LIN {X 0,Y 488.826,Z 251.849,A -85,B 0,C 180,E1 23621.041,E2 23621.041} C_VEL
LIN {X 0,Y 488.773,Z 251.852,A -85,B 0,C 180,E1 23617.658,E2 23617.658} C_VEL
LIN {X 0,Y 488.76,Z 251.853,A -85,B 0,C 180,E1 23614.093,E2 23614.093} C_VEL
LIN {X 0,Y 488.789,Z 251.852,A -85,B 0,C 180,E1 23610.622,E2 23610.622} C_VEL
LIN {X 0,Y 488.787,Z 251.853,A -85,B 0,C 180,E1 23607.273,E2 23607.273} C_VEL
LIN {X 0,Y 488.779,Z 251.938,A -85,B 0,C 180,E1 23606.334,E2 23606.334} C_VEL
LIN {X 0,Y 489.957,Z 255.178,A -85,B 0,C 180,E1 23606.114,E2 23606.114} C_VEL
LIN {X 0,Y 492.29,Z 257.974,A -85,B 0,C 180,E1 23605.77,E2 23605.77} C_VEL
LIN {X 0,Y 494.97,Z 261.991,A -85,B 0,C 180,E1 23605.374,E2 23605.374} C_VEL
LIN {X 0,Y 505.952,Z 279.714,A -85,B 0,C 180,E1 23603.9,E2 23603.9} C_VEL
LIN {X 0,Y 508.929,Z 284.891,A -85,B 0,C 180,E1 23603.527,E2 23603.527} C_VEL
LIN {X 0,Y 506.243,Z 428.401,A -85,B 0,C 180,E1 23601.176,E2 23601.176} C_VEL
LIN {X 0,Y 504.683,Z 530.578,A -85,B 0,C 180,E1 23599.559,E2 23599.559} C_VEL
LIN {X 0,Y 503.855,Z 552.45,A -85,B 0,C 180,E1 23599.012,E2 23599.012} C_VEL
LIN {X 0,Y 502.715,Z 574.756,A -85,B 0,C 180,E1 23598.227,E2 23598.227} C_VEL
LIN {X 0,Y 501.313,Z 596.319,A -85,B 0,C 180,E1 23597.229,E2 23597.229} C_VEL
LIN {X 0,Y 499.603,Z 617.696,A -85,B 0,C 180,E1 23595.974,E2 23595.974} C_VEL
LIN {X 0,Y 497.826,Z 637.974,A -85,B 0,C 180,E1 23594.516,E2 23594.516} C_VEL
LIN {X 0,Y 496.107,Z 656.509,A -85,B 0,C 180,E1 23592.928,E2 23592.928} C_VEL
LIN {X 0,Y 494.361,Z 674.873,A -85,B 0,C 180,E1 23591.079,E2 23591.079} C_VEL
LIN {X 0,Y 492.804,Z 691.473,A -85,B 0,C 180,E1 23589.107,E2 23589.107} C_VEL
LIN {X 0,Y 491.464,Z 706.623,A -85,B 0,C 180,E1 23587.013,E2 23587.013} C_VEL
LIN {X 0,Y 490.28,Z 720.943,A -85,B 0,C 180,E1 23584.681,E2 23584.681} C_VEL
LIN {X 0,Y 489.411,Z 733.128,A -85,B 0,C 180,E1 23582.343,E2 23582.343} C_VEL
LIN {X 0,Y 488.737,Z 744.343,A -85,B 0,C 180,E1 23579.767,E2 23579.767} C_VEL
LIN {X 0,Y 488.322,Z 753.138,A -85,B 0,C 180,E1 23577.302,E2 23577.302} C_VEL
LIN {X 0,Y 488.079,Z 760.481,A -85,B 0,C 180,E1 23574.712,E2 23574.712} C_VEL
LIN {X 0,Y 487.958,Z 765.848,A -85,B 0,C 180,E1 23572.229,E2 23572.229} C_VEL
LIN {X 0,Y 487.912,Z 769.627,A -85,B 0,C 180,E1 23569.732,E2 23569.732} C_VEL
LIN {X 0,Y 487.912,Z 771.838,A -85,B 0,C 180,E1 23567.215,E2 23567.215} C_VEL
LIN {X 0,Y 487.904,Z 772.465,A -85,B 0,C 180,E1 23564.673,E2 23564.673} C_VEL
LIN {X 0,Y 487.91,Z 771.462,A -85,B 0,C 180,E1 23562.1,E2 23562.1} C_VEL
LIN {X 0,Y 487.918,Z 768.918,A -85,B 0,C 180,E1 23559.615,E2 23559.615} C_VEL
LIN {X 0,Y 487.984,Z 764.727,A -85,B 0,C 180,E1 23557.091,E2 23557.091} C_VEL
LIN {X 0,Y 488.128,Z 758.759,A -85,B 0,C 180,E1 23554.525,E2 23554.525} C_VEL
LIN {X 0,Y 488.397,Z 751.272,A -85,B 0,C 180,E1 23552.045,E2 23552.045} C_VEL
LIN {X 0,Y 488.888,Z 741.478,A -85,B 0,C 180,E1 23549.432,E2 23549.432} C_VEL
LIN {X 0,Y 489.602,Z 730.156,A -85,B 0,C 180,E1 23546.96,E2 23546.96} C_VEL
LIN {X 0,Y 490.56,Z 717.417,A -85,B 0,C 180,E1 23544.616,E2 23544.616} C_VEL
LIN {X 0,Y 491.761,Z 702.995,A -85,B 0,C 180,E1 23542.37,E2 23542.37} C_VEL
LIN {X 0,Y 493.172,Z 687.603,A -85,B 0,C 180,E1 23540.313,E2 23540.313} C_VEL
LIN {X 0,Y 494.808,Z 670.219,A -85,B 0,C 180,E1 23538.336,E2 23538.336} C_VEL
LIN {X 0,Y 496.461,Z 652.681,A -85,B 0,C 180,E1 23536.629,E2 23536.629} C_VEL
LIN {X 0,Y 498.323,Z 632.595,A -85,B 0,C 180,E1 23534.982,E2 23534.982} C_VEL
LIN {X 0,Y 500.016,Z 612.711,A -85,B 0,C 180,E1 23533.621,E2 23533.621} C_VEL
LIN {X 0,Y 501.553,Z 593.125,A -85,B 0,C 180,E1 23532.517,E2 23532.517} C_VEL
LIN {X 0,Y 502.952,Z 571.382,A -85,B 0,C 180,E1 23531.536,E2 23531.536} C_VEL
LIN {X 0,Y 503.202,Z 567.217,A -85,B 0,C 180,E1 23531.379,E2 23531.379} C_VEL
LIN {X 0,Y 502.78,Z 559.985,A -85,B 0,C 180,E1 23531.059,E2 23531.059} C_VEL
LIN {X 0,Y 498.556,Z 542.003,A -85,B 0,C 180,E1 23530.149,E2 23530.149} C_VEL
LIN {X 0,Y 497.979,Z 534.584,A -85,B 0,C 180,E1 23529.907,E2 23529.907} C_VEL
LIN {X 0,Y 498.643,Z 507.178,A -85,B 0,C 180,E1 23529.418,E2 23529.418} C_VEL
LIN {X 0,Y 501.545,Z 350.429,A -85,B 0,C 180,E1 23526.864,E2 23526.864} C_VEL
LIN {X 0,Y 502.677,Z 287.585,A -85,B 0,C 180,E1 23525.824,E2 23525.824} C_VEL
LIN {X 0,Y 489.417,Z 266.799,A -85,B 0,C 180,E1 23524.129,E2 23524.129} C_VEL
LIN {X 0,Y 484.118,Z 258.644,A -85,B 0,C 180,E1 23523.414,E2 23523.414} C_VEL
LIN {X 0,Y 481.453,Z 254.949,A -85,B 0,C 180,E1 23523.053,E2 23523.053} C_VEL
LIN {X 0,Y 480.884,Z 252.838,A -85,B 0,C 180,E1 23522.938,E2 23522.938} C_VEL
LIN {X 0,Y 480.896,Z 252.835,A -85,B 0,C 180,E1 23519.386,E2 23519.386} C_VEL
LIN {X 0,Y 480.859,Z 252.836,A -85,B 0,C 180,E1 23515.892,E2 23515.892} C_VEL
LIN {X 0,Y 480.851,Z 252.838,A -85,B 0,C 180,E1 23512.238,E2 23512.238} C_VEL
LIN {X 0,Y 480.877,Z 252.834,A -85,B 0,C 180,E1 23508.676,E2 23508.676} C_VEL
LIN {X 0,Y 480.896,Z 252.833,A -85,B 0,C 180,E1 23505.065,E2 23505.065} C_VEL
LIN {X 0,Y 480.863,Z 252.833,A -85,B 0,C 180,E1 23501.515,E2 23501.515} C_VEL
LIN {X 0,Y 480.847,Z 252.834,A -85,B 0,C 180,E1 23498.009,E2 23498.009} C_VEL
LIN {X 0,Y 480.877,Z 252.835,A -85,B 0,C 180,E1 23494.533,E2 23494.533} C_VEL
LIN {X 0,Y 480.891,Z 252.83,A -85,B 0,C 180,E1 23490.954,E2 23490.954} C_VEL
LIN {X 0,Y 480.848,Z 252.833,A -85,B 0,C 180,E1 23487.498,E2 23487.498} C_VEL
LIN {X 0,Y 480.844,Z 252.834,A -85,B 0,C 180,E1 23483.914,E2 23483.914} C_VEL
LIN {X 0,Y 480.88,Z 252.836,A -85,B 0,C 180,E1 23480.426,E2 23480.426} C_VEL
LIN {X 0,Y 480.875,Z 252.831,A -85,B 0,C 180,E1 23476.902,E2 23476.902} C_VEL
LIN {X 0,Y 480.838,Z 252.834,A -85,B 0,C 180,E1 23473.447,E2 23473.447} C_VEL
LIN {X 0,Y 480.843,Z 252.835,A -85,B 0,C 180,E1 23469.809,E2 23469.809} C_VEL
LIN {X 0,Y 480.887,Z 252.831,A -85,B 0,C 180,E1 23466.343,E2 23466.343} C_VEL
LIN {X 0,Y 480.864,Z 252.835,A -85,B 0,C 180,E1 23462.779,E2 23462.779} C_VEL
LIN {X 0,Y 480.832,Z 252.838,A -85,B 0,C 180,E1 23459.374,E2 23459.374} C_VEL
LIN {X 0,Y 480.854,Z 252.84,A -85,B 0,C 180,E1 23455.846,E2 23455.846} C_VEL
LIN {X 0,Y 480.888,Z 252.831,A -85,B 0,C 180,E1 23452.32,E2 23452.32} C_VEL
LIN {X 0,Y 480.84,Z 252.835,A -85,B 0,C 180,E1 23448.824,E2 23448.824} C_VEL
LIN {X 0,Y 480.83,Z 252.838,A -85,B 0,C 180,E1 23445.326,E2 23445.326} C_VEL
LIN {X 0,Y 480.868,Z 252.841,A -85,B 0,C 180,E1 23441.867,E2 23441.867} C_VEL
LIN {X 0,Y 480.859,Z 252.833,A -85,B 0,C 180,E1 23438.384,E2 23438.384} C_VEL
LIN {X 0,Y 480.823,Z 252.833,A -85,B 0,C 180,E1 23434.877,E2 23434.877} C_VEL
LIN {X 0,Y 480.828,Z 252.836,A -85,B 0,C 180,E1 23431.282,E2 23431.282} C_VEL
LIN {X 0,Y 480.885,Z 252.838,A -85,B 0,C 180,E1 23427.89,E2 23427.89} C_VEL
LIN {X 0,Y 480.84,Z 252.835,A -85,B 0,C 180,E1 23424.311,E2 23424.311} C_VEL
LIN {X 0,Y 480.817,Z 252.836,A -85,B 0,C 180,E1 23420.828,E2 23420.828} C_VEL
LIN {X 0,Y 480.837,Z 252.838,A -85,B 0,C 180,E1 23417.297,E2 23417.297} C_VEL
LIN {X 0,Y 480.87,Z 252.834,A -85,B 0,C 180,E1 23413.832,E2 23413.832} C_VEL
LIN {X 0,Y 480.82,Z 252.836,A -85,B 0,C 180,E1 23410.3,E2 23410.3} C_VEL
LIN {X 0,Y 480.813,Z 252.838,A -85,B 0,C 180,E1 23406.806,E2 23406.806} C_VEL
LIN {X 0,Y 480.853,Z 252.839,A -85,B 0,C 180,E1 23403.336,E2 23403.336} C_VEL
LIN {X 0,Y 480.839,Z 252.836,A -85,B 0,C 180,E1 23399.879,E2 23399.879} C_VEL
LIN {X 0,Y 480.812,Z 252.839,A -85,B 0,C 180,E1 23396.422,E2 23396.422} C_VEL
LIN {X 0,Y 480.834,Z 252.839,A -85,B 0,C 180,E1 23392.951,E2 23392.951} C_VEL
LIN {X 0,Y 480.87,Z 252.837,A -85,B 0,C 180,E1 23389.456,E2 23389.456} C_VEL
LIN {X 0,Y 480.823,Z 252.837,A -85,B 0,C 180,E1 23386.04,E2 23386.04} C_VEL
LIN {X 0,Y 480.821,Z 252.838,A -85,B 0,C 180,E1 23382.45,E2 23382.45} C_VEL
LIN {X 0,Y 480.866,Z 252.834,A -85,B 0,C 180,E1 23378.998,E2 23378.998} C_VEL
LIN {X 0,Y 480.849,Z 252.837,A -85,B 0,C 180,E1 23375.556,E2 23375.556} C_VEL
LIN {X 0,Y 480.822,Z 252.837,A -85,B 0,C 180,E1 23372.097,E2 23372.097} C_VEL
LIN {X 0,Y 480.853,Z 252.837,A -85,B 0,C 180,E1 23368.678,E2 23368.678} C_VEL
LIN {X 0,Y 480.879,Z 252.835,A -85,B 0,C 180,E1 23365.124,E2 23365.124} C_VEL
LIN {X 0,Y 480.837,Z 252.839,A -85,B 0,C 180,E1 23361.62,E2 23361.62} C_VEL
LIN {X 0,Y 480.833,Z 252.842,A -85,B 0,C 180,E1 23358.108,E2 23358.108} C_VEL
LIN {X 0,Y 480.893,Z 252.932,A -85,B 0,C 180,E1 23356.746,E2 23356.746} C_VEL
LIN {X 0,Y 482.026,Z 256.137,A -85,B 0,C 180,E1 23356.311,E2 23356.311} C_VEL
LIN {X 0,Y 486.724,Z 266.041,A -85,B 0,C 180,E1 23354.868,E2 23354.868} C_VEL
LIN {X 0,Y 494.252,Z 282.954,A -85,B 0,C 180,E1 23352.577,E2 23352.577} C_VEL
LIN {X 0,Y 498.97,Z 294.265,A -85,B 0,C 180,E1 23351.153,E2 23351.153} C_VEL
LIN {X 0,Y 498.76,Z 300.518,A -85,B 0,C 180,E1 23350.689,E2 23350.689} C_VEL
LIN {X 0,Y 503.225,Z 328.094,A -85,B 0,C 180,E1 23349.716,E2 23349.716} C_VEL
LIN {X 0,Y 499.682,Z 515.938,A -85,B 0,C 180,E1 23346.648,E2 23346.648} C_VEL
LIN {X 0,Y 498.054,Z 606.169,A -85,B 0,C 180,E1 23345.186,E2 23345.186} C_VEL
LIN {X 0,Y 497.13,Z 628.175,A -85,B 0,C 180,E1 23344.647,E2 23344.647} C_VEL
LIN {X 0,Y 495.947,Z 649.87,A -85,B 0,C 180,E1 23343.911,E2 23343.911} C_VEL
LIN {X 0,Y 494.532,Z 671.447,A -85,B 0,C 180,E1 23342.958,E2 23342.958} C_VEL
LIN {X 0,Y 492.943,Z 691.876,A -85,B 0,C 180,E1 23341.826,E2 23341.826} C_VEL
LIN {X 0,Y 491.226,Z 712.419,A -85,B 0,C 180,E1 23340.451,E2 23340.451} C_VEL
LIN {X 0,Y 489.577,Z 729.553,A -85,B 0,C 180,E1 23339.061,E2 23339.061} C_VEL
LIN {X 0,Y 487.819,Z 746.483,A -85,B 0,C 180,E1 23337.439,E2 23337.439} C_VEL
LIN {X 0,Y 486.065,Z 763.653,A -85,B 0,C 180,E1 23335.526,E2 23335.526} C_VEL
LIN {X 0,Y 484.507,Z 779.487,A -85,B 0,C 180,E1 23333.469,E2 23333.469} C_VEL
LIN {X 0,Y 483.123,Z 794.1,A -85,B 0,C 180,E1 23331.232,E2 23331.232} C_VEL
LIN {X 0,Y 482.039,Z 806.869,A -85,B 0,C 180,E1 23328.941,E2 23328.941} C_VEL
LIN {X 0,Y 481.203,Z 818.27,A -85,B 0,C 180,E1 23326.537,E2 23326.537} C_VEL
LIN {X 0,Y 480.621,Z 827.976,A -85,B 0,C 180,E1 23324.086,E2 23324.086} C_VEL
LIN {X 0,Y 480.255,Z 835.826,A -85,B 0,C 180,E1 23321.649,E2 23321.649} C_VEL
LIN {X 0,Y 480.045,Z 842.385,A -85,B 0,C 180,E1 23319.107,E2 23319.107} C_VEL
LIN {X 0,Y 479.949,Z 847.021,A -85,B 0,C 180,E1 23316.698,E2 23316.698} C_VEL
LIN {X 0,Y 479.913,Z 850.447,A -85,B 0,C 180,E1 23314.061,E2 23314.061} C_VEL
LIN {X 0,Y 479.898,Z 852.21,A -85,B 0,C 180,E1 23311.551,E2 23311.551} C_VEL
LIN {X 0,Y 479.91,Z 852.326,A -85,B 0,C 180,E1 23309.044,E2 23309.044} C_VEL
LIN {X 0,Y 479.909,Z 850.897,A -85,B 0,C 180,E1 23306.415,E2 23306.415} C_VEL
LIN {X 0,Y 479.935,Z 848.137,A -85,B 0,C 180,E1 23304.02,E2 23304.02} C_VEL
LIN {X 0,Y 480.008,Z 843.65,A -85,B 0,C 180,E1 23301.494,E2 23301.494} C_VEL
LIN {X 0,Y 480.176,Z 837.933,A -85,B 0,C 180,E1 23299.076,E2 23299.076} C_VEL
LIN {X 0,Y 480.484,Z 830.473,A -85,B 0,C 180,E1 23296.644,E2 23296.644} C_VEL
LIN {X 0,Y 481.033,Z 820.833,A -85,B 0,C 180,E1 23294.075,E2 23294.075} C_VEL
LIN {X 0,Y 481.779,Z 810.346,A -85,B 0,C 180,E1 23291.736,E2 23291.736} C_VEL
LIN {X 0,Y 482.795,Z 797.753,A -85,B 0,C 180,E1 23289.385,E2 23289.385} C_VEL
LIN {X 0,Y 484.073,Z 783.703,A -85,B 0,C 180,E1 23287.149,E2 23287.149} C_VEL
LIN {X 0,Y 485.611,Z 768.194,A -85,B 0,C 180,E1 23285.033,E2 23285.033} C_VEL
LIN {X 0,Y 487.338,Z 751.503,A -85,B 0,C 180,E1 23283.081,E2 23283.081} C_VEL
LIN {X 0,Y 489.084,Z 734.081,A -85,B 0,C 180,E1 23281.353,E2 23281.353} C_VEL
LIN {X 0,Y 490.931,Z 715.707,A -85,B 0,C 180,E1 23279.797,E2 23279.797} C_VEL
LIN {X 0,Y 492.168,Z 700.762,A -85,B 0,C 180,E1 23278.749,E2 23278.749} C_VEL
LIN {X 0,Y 493.688,Z 680.03,A -85,B 0,C 180,E1 23277.54,E2 23277.54} C_VEL
LIN {X 0,Y 495.09,Z 659.096,A -85,B 0,C 180,E1 23276.54,E2 23276.54} C_VEL
LIN {X 0,Y 496.257,Z 636.725,A -85,B 0,C 180,E1 23275.709,E2 23275.709} C_VEL
LIN {X 0,Y 497.248,Z 614.263,A -85,B 0,C 180,E1 23275.096,E2 23275.096} C_VEL
LIN {X 0,Y 497.876,Z 589.797,A -85,B 0,C 180,E1 23274.643,E2 23274.643} C_VEL
LIN {X 0,Y 500.406,Z 423.697,A -85,B 0,C 180,E1 23272.015,E2 23272.015} C_VEL
LIN {X 0,Y 502.407,Z 326.034,A -85,B 0,C 180,E1 23270.334,E2 23270.334} C_VEL
LIN {X 0,Y 497.215,Z 292.664,A -85,B 0,C 180,E1 23269.123,E2 23269.123} C_VEL
LIN {X 0,Y 488.051,Z 269.345,A -85,B 0,C 180,E1 23266.234,E2 23266.234} C_VEL
LIN {X 0,Y 483.81,Z 259.793,A -85,B 0,C 180,E1 23264.808,E2 23264.808} C_VEL
LIN {X 0,Y 482.417,Z 256.717,A -85,B 0,C 180,E1 23264.305,E2 23264.305} C_VEL
LIN {X 0,Y 480.922,Z 253.362,A -85,B 0,C 180,E1 23263.732,E2 23263.732} C_VEL
LIN {X 0,Y 480.845,Z 252.841,A -85,B 0,C 180,E1 23263.645,E2 23263.645} C_VEL
LIN {X 0,Y 480.825,Z 252.843,A -85,B 0,C 180,E1 23260.139,E2 23260.139} C_VEL
LIN {X 0,Y 480.863,Z 252.84,A -85,B 0,C 180,E1 23256.788,E2 23256.788} C_VEL
LIN {X 0,Y 480.858,Z 252.839,A -85,B 0,C 180,E1 23253.291,E2 23253.291} C_VEL
LIN {X 0,Y 480.818,Z 252.844,A -85,B 0,C 180,E1 23249.87,E2 23249.87} C_VEL
LIN {X 0,Y 480.877,Z 253.089,A -85,B 0,C 180,E1 23247.326,E2 23247.326} C_VEL
LIN {X 0,Y 482.124,Z 256.249,A -85,B 0,C 180,E1 23247.067,E2 23247.067} C_VEL
LIN {X 0,Y 484.497,Z 259.065,A -85,B 0,C 180,E1 23246.672,E2 23246.672} C_VEL
LIN {X 0,Y 487.154,Z 263.069,A -85,B 0,C 180,E1 23246.243,E2 23246.243} C_VEL
LIN {X 0,Y 493.728,Z 273.293,A -85,B 0,C 180,E1 23245.247,E2 23245.247} C_VEL
LIN {X 0,Y 502.608,Z 287.934,A -85,B 0,C 180,E1 23244.046,E2 23244.046} C_VEL
LIN {X 0,Y 499.77,Z 411.695,A -85,B 0,C 180,E1 23241.94,E2 23241.94} C_VEL
LIN {X 0,Y 497.748,Z 532.141,A -85,B 0,C 180,E1 23239.996,E2 23239.996} C_VEL
LIN {X 0,Y 496.86,Z 554.258,A -85,B 0,C 180,E1 23239.428,E2 23239.428} C_VEL
LIN {X 0,Y 495.706,Z 575.864,A -85,B 0,C 180,E1 23238.651,E2 23238.651} C_VEL
LIN {X 0,Y 494.28,Z 596.991,A -85,B 0,C 180,E1 23237.665,E2 23237.665} C_VEL
LIN {X 0,Y 492.582,Z 617.72,A -85,B 0,C 180,E1 23236.45,E2 23236.45} C_VEL
LIN {X 0,Y 490.853,Z 636.705,A -85,B 0,C 180,E1 23235.086,E2 23235.086} C_VEL
LIN {X 0,Y 488.972,Z 655.448,A -85,B 0,C 180,E1 23233.481,E2 23233.481} C_VEL
LIN {X 0,Y 487.012,Z 674.481,A -85,B 0,C 180,E1 23231.548,E2 23231.548} C_VEL
LIN {X 0,Y 485.37,Z 690.695,A -85,B 0,C 180,E1 23229.607,E2 23229.607} C_VEL
LIN {X 0,Y 483.813,Z 706.737,A -85,B 0,C 180,E1 23227.363,E2 23227.363} C_VEL
LIN {X 0,Y 482.52,Z 721.036,A -85,B 0,C 180,E1 23224.994,E2 23224.994} C_VEL
LIN {X 0,Y 481.565,Z 733.206,A -85,B 0,C 180,E1 23222.62,E2 23222.62} C_VEL
LIN {X 0,Y 480.827,Z 744.4,A -85,B 0,C 180,E1 23220.002,E2 23220.002} C_VEL
LIN {X 0,Y 480.368,Z 753.178,A -85,B 0,C 180,E1 23217.496,E2 23217.496} C_VEL
LIN {X 0,Y 480.094,Z 760.514,A -85,B 0,C 180,E1 23214.864,E2 23214.864} C_VEL
LIN {X 0,Y 479.967,Z 765.868,A -85,B 0,C 180,E1 23212.34,E2 23212.34} C_VEL
LIN {X 0,Y 479.912,Z 769.638,A -85,B 0,C 180,E1 23209.802,E2 23209.802} C_VEL
LIN {X 0,Y 479.912,Z 771.885,A -85,B 0,C 180,E1 23207.174,E2 23207.174} C_VEL
LIN {X 0,Y 479.904,Z 772.464,A -85,B 0,C 180,E1 23204.659,E2 23204.659} C_VEL
LIN {X 0,Y 479.91,Z 771.454,A -85,B 0,C 180,E1 23202.042,E2 23202.042} C_VEL
LIN {X 0,Y 479.922,Z 768.906,A -85,B 0,C 180,E1 23199.514,E2 23199.514} C_VEL
LIN {X 0,Y 479.997,Z 764.701,A -85,B 0,C 180,E1 23196.947,E2 23196.947} C_VEL
LIN {X 0,Y 480.151,Z 758.725,A -85,B 0,C 180,E1 23194.336,E2 23194.336} C_VEL
LIN {X 0,Y 480.455,Z 751.222,A -85,B 0,C 180,E1 23191.812,E2 23191.812} C_VEL
LIN {X 0,Y 481.008,Z 741.388,A -85,B 0,C 180,E1 23189.149,E2 23189.149} C_VEL
LIN {X 0,Y 481.796,Z 730.063,A -85,B 0,C 180,E1 23186.639,E2 23186.639} C_VEL
LIN {X 0,Y 482.837,Z 717.379,A -85,B 0,C 180,E1 23184.268,E2 23184.268} C_VEL
LIN {X 0,Y 484.19,Z 702.534,A -85,B 0,C 180,E1 23181.927,E2 23181.927} C_VEL
LIN {X 0,Y 485.697,Z 687.44,A -85,B 0,C 180,E1 23179.887,E2 23179.887} C_VEL
LIN {X 0,Y 487.48,Z 670.032,A -85,B 0,C 180,E1 23177.882,E2 23177.882} C_VEL
LIN {X 0,Y 489.27,Z 652.463,A -85,B 0,C 180,E1 23176.154,E2 23176.154} C_VEL
LIN {X 0,Y 491.276,Z 632.355,A -85,B 0,C 180,E1 23174.487,E2 23174.487} C_VEL
LIN {X 0,Y 493.103,Z 612.202,A -85,B 0,C 180,E1 23173.105,E2 23173.105} C_VEL
LIN {X 0,Y 494.76,Z 591.707,A -85,B 0,C 180,E1 23171.957,E2 23171.957} C_VEL
LIN {X 0,Y 496.194,Z 570.406,A -85,B 0,C 180,E1 23171.005,E2 23171.005} C_VEL
LIN {X 0,Y 497.395,Z 548.543,A -85,B 0,C 180,E1 23170.264,E2 23170.264} C_VEL
LIN {X 0,Y 497.979,Z 534.584,A -85,B 0,C 180,E1 23169.907,E2 23169.907} C_VEL
LIN {X 0,Y 497.434,Z 527.084,A -85,B 0,C 180,E1 23169.683,E2 23169.683} C_VEL
LIN {X 0,Y 492.603,Z 507.384,A -85,B 0,C 180,E1 23168.951,E2 23168.951} C_VEL
LIN {X 0,Y 492.087,Z 500.873,A -85,B 0,C 180,E1 23168.801,E2 23168.801} C_VEL
LIN {X 0,Y 495.963,Z 317.795,A -85,B 0,C 180,E1 23165.755,E2 23165.755} C_VEL
LIN {X 0,Y 496.395,Z 290.909,A -85,B 0,C 180,E1 23165.299,E2 23165.299} C_VEL
LIN {X 0,Y 484.26,Z 271.876,A -85,B 0,C 180,E1 23163.704,E2 23163.704} C_VEL
LIN {X 0,Y 477.954,Z 262.595,A -85,B 0,C 180,E1 23162.844,E2 23162.844} C_VEL
LIN {X 0,Y 475.512,Z 258.789,A -85,B 0,C 180,E1 23162.497,E2 23162.497} C_VEL
LIN {X 0,Y 473.393,Z 255.718,A -85,B 0,C 180,E1 23162.194,E2 23162.194} C_VEL
LIN {X 0,Y 472.921,Z 253.828,A -85,B 0,C 180,E1 23162.087,E2 23162.087} C_VEL
LIN {X 0,Y 472.92,Z 253.828,A -85,B 0,C 180,E1 23158.406,E2 23158.406} C_VEL
LIN {X 0,Y 472.948,Z 253.822,A -85,B 0,C 180,E1 23154.88,E2 23154.88} C_VEL
LIN {X 0,Y 472.96,Z 253.821,A -85,B 0,C 180,E1 23151.193,E2 23151.193} C_VEL
LIN {X 0,Y 472.93,Z 253.823,A -85,B 0,C 180,E1 23147.552,E2 23147.552} C_VEL
LIN {X 0,Y 472.91,Z 253.82,A -85,B 0,C 180,E1 23143.948,E2 23143.948} C_VEL
LIN {X 0,Y 472.922,Z 253.827,A -85,B 0,C 180,E1 23140.354,E2 23140.354} C_VEL
LIN {X 0,Y 472.958,Z 253.823,A -85,B 0,C 180,E1 23136.8,E2 23136.8} C_VEL
LIN {X 0,Y 472.937,Z 253.821,A -85,B 0,C 180,E1 23133.152,E2 23133.152} C_VEL
LIN {X 0,Y 472.906,Z 253.82,A -85,B 0,C 180,E1 23129.638,E2 23129.638} C_VEL
LIN {X 0,Y 472.907,Z 253.817,A -85,B 0,C 180,E1 23126,E2 23126} C_VEL
LIN {X 0,Y 472.946,Z 253.818,A -85,B 0,C 180,E1 23122.47,E2 23122.47} C_VEL
LIN {X 0,Y 472.938,Z 253.821,A -85,B 0,C 180,E1 23118.909,E2 23118.909} C_VEL
LIN {X 0,Y 472.901,Z 253.823,A -85,B 0,C 180,E1 23115.429,E2 23115.429} C_VEL
LIN {X 0,Y 472.904,Z 253.824,A -85,B 0,C 180,E1 23111.766,E2 23111.766} C_VEL
LIN {X 0,Y 472.946,Z 253.827,A -85,B 0,C 180,E1 23108.288,E2 23108.288} C_VEL
LIN {X 0,Y 472.933,Z 253.821,A -85,B 0,C 180,E1 23104.721,E2 23104.721} C_VEL
LIN {X 0,Y 472.897,Z 253.822,A -85,B 0,C 180,E1 23101.181,E2 23101.181} C_VEL
LIN {X 0,Y 472.896,Z 253.821,A -85,B 0,C 180,E1 23097.519,E2 23097.519} C_VEL
LIN {X 0,Y 472.928,Z 253.823,A -85,B 0,C 180,E1 23094.005,E2 23094.005} C_VEL
LIN {X 0,Y 472.934,Z 253.826,A -85,B 0,C 180,E1 23090.481,E2 23090.481} C_VEL
LIN {X 0,Y 472.891,Z 253.827,A -85,B 0,C 180,E1 23087.014,E2 23087.014} C_VEL
LIN {X 0,Y 472.891,Z 253.826,A -85,B 0,C 180,E1 23083.339,E2 23083.339} C_VEL
LIN {X 0,Y 472.927,Z 253.822,A -85,B 0,C 180,E1 23079.833,E2 23079.833} C_VEL
LIN {X 0,Y 472.924,Z 253.828,A -85,B 0,C 180,E1 23076.294,E2 23076.294} C_VEL
LIN {X 0,Y 472.886,Z 253.828,A -85,B 0,C 180,E1 23072.768,E2 23072.768} C_VEL
LIN {X 0,Y 472.884,Z 253.826,A -85,B 0,C 180,E1 23069.096,E2 23069.096} C_VEL
LIN {X 0,Y 472.926,Z 253.821,A -85,B 0,C 180,E1 23065.682,E2 23065.682} C_VEL
LIN {X 0,Y 472.917,Z 253.826,A -85,B 0,C 180,E1 23062.104,E2 23062.104} C_VEL
LIN {X 0,Y 472.878,Z 253.827,A -85,B 0,C 180,E1 23058.617,E2 23058.617} C_VEL
LIN {X 0,Y 472.878,Z 253.826,A -85,B 0,C 180,E1 23054.928,E2 23054.928} C_VEL
LIN {X 0,Y 472.917,Z 253.825,A -85,B 0,C 180,E1 23051.461,E2 23051.461} C_VEL
LIN {X 0,Y 472.911,Z 253.829,A -85,B 0,C 180,E1 23047.897,E2 23047.897} C_VEL
LIN {X 0,Y 472.871,Z 253.828,A -85,B 0,C 180,E1 23044.485,E2 23044.485} C_VEL
LIN {X 0,Y 472.878,Z 253.825,A -85,B 0,C 180,E1 23040.846,E2 23040.846} C_VEL
LIN {X 0,Y 472.929,Z 253.824,A -85,B 0,C 180,E1 23037.454,E2 23037.454} C_VEL
LIN {X 0,Y 472.892,Z 253.825,A -85,B 0,C 180,E1 23033.93,E2 23033.93} C_VEL
LIN {X 0,Y 472.877,Z 253.828,A -85,B 0,C 180,E1 23030.383,E2 23030.383} C_VEL
LIN {X 0,Y 472.896,Z 253.825,A -85,B 0,C 180,E1 23026.799,E2 23026.799} C_VEL
LIN {X 0,Y 472.931,Z 253.823,A -85,B 0,C 180,E1 23023.415,E2 23023.415} C_VEL
LIN {X 0,Y 472.893,Z 253.827,A -85,B 0,C 180,E1 23019.84,E2 23019.84} C_VEL
LIN {X 0,Y 472.885,Z 253.825,A -85,B 0,C 180,E1 23016.276,E2 23016.276} C_VEL
LIN {X 0,Y 472.922,Z 253.823,A -85,B 0,C 180,E1 23012.826,E2 23012.826} C_VEL
LIN {X 0,Y 472.921,Z 253.828,A -85,B 0,C 180,E1 23009.367,E2 23009.367} C_VEL
LIN {X 0,Y 472.888,Z 253.83,A -85,B 0,C 180,E1 23005.922,E2 23005.922} C_VEL
LIN {X 0,Y 472.896,Z 253.826,A -85,B 0,C 180,E1 23002.254,E2 23002.254} C_VEL
LIN {X 0,Y 472.947,Z 253.826,A -85,B 0,C 180,E1 22998.815,E2 22998.815} C_VEL
LIN {X 0,Y 472.912,Z 253.941,A -85,B 0,C 180,E1 22997.588,E2 22997.588} C_VEL
LIN {X 0,Y 474.308,Z 257.409,A -85,B 0,C 180,E1 22997.085,E2 22997.085} C_VEL
LIN {X 0,Y 482.059,Z 273.946,A -85,B 0,C 180,E1 22994.648,E2 22994.648} C_VEL
LIN {X 0,Y 490.751,Z 294.314,A -85,B 0,C 180,E1 22991.931,E2 22991.931} C_VEL
LIN {X 0,Y 492.197,Z 298.048,A -85,B 0,C 180,E1 22991.469,E2 22991.469} C_VEL
LIN {X 0,Y 492.304,Z 300.443,A -85,B 0,C 180,E1 22991.326,E2 22991.326} C_VEL
LIN {X 0,Y 496.987,Z 329.547,A -85,B 0,C 180,E1 22990.275,E2 22990.275} C_VEL
LIN {X 0,Y 492.643,Z 539.067,A -85,B 0,C 180,E1 22986.799,E2 22986.799} C_VEL
LIN {X 0,Y 491.203,Z 608.625,A -85,B 0,C 180,E1 22985.632,E2 22985.632} C_VEL
LIN {X 0,Y 490.172,Z 630.155,A -85,B 0,C 180,E1 22985.073,E2 22985.073} C_VEL
LIN {X 0,Y 488.787,Z 652.65,A -85,B 0,C 180,E1 22984.267,E2 22984.267} C_VEL
LIN {X 0,Y 487.271,Z 673.754,A -85,B 0,C 180,E1 22983.29,E2 22983.29} C_VEL
LIN {X 0,Y 485.608,Z 693.572,A -85,B 0,C 180,E1 22982.156,E2 22982.156} C_VEL
LIN {X 0,Y 483.783,Z 713.671,A -85,B 0,C 180,E1 22980.763,E2 22980.763} C_VEL
LIN {X 0,Y 481.903,Z 732.987,A -85,B 0,C 180,E1 22979.18,E2 22979.18} C_VEL
LIN {X 0,Y 480.419,Z 747.492,A -85,B 0,C 180,E1 22977.786,E2 22977.786} C_VEL
LIN {X 0,Y 478.521,Z 764.665,A -85,B 0,C 180,E1 22975.825,E2 22975.825} C_VEL
LIN {X 0,Y 476.945,Z 779.488,A -85,B 0,C 180,E1 22973.864,E2 22973.864} C_VEL
LIN {X 0,Y 475.467,Z 793.778,A -85,B 0,C 180,E1 22971.645,E2 22971.645} C_VEL
LIN {X 0,Y 474.28,Z 806.552,A -85,B 0,C 180,E1 22969.327,E2 22969.327} C_VEL
LIN {X 0,Y 473.361,Z 817.974,A -85,B 0,C 180,E1 22966.892,E2 22966.892} C_VEL
LIN {X 0,Y 472.719,Z 827.516,A -85,B 0,C 180,E1 22964.451,E2 22964.451} C_VEL
LIN {X 0,Y 472.306,Z 835.472,A -85,B 0,C 180,E1 22961.972,E2 22961.972} C_VEL
LIN {X 0,Y 472.074,Z 842.131,A -85,B 0,C 180,E1 22959.385,E2 22959.385} C_VEL
LIN {X 0,Y 471.964,Z 846.815,A -85,B 0,C 180,E1 22956.934,E2 22956.934} C_VEL
LIN {X 0,Y 471.917,Z 850.333,A -85,B 0,C 180,E1 22954.251,E2 22954.251} C_VEL
LIN {X 0,Y 471.902,Z 852.085,A -85,B 0,C 180,E1 22951.82,E2 22951.82} C_VEL
LIN {X 0,Y 471.902,Z 852.371,A -85,B 0,C 180,E1 22949.27,E2 22949.27} C_VEL
LIN {X 0,Y 471.915,Z 851.234,A -85,B 0,C 180,E1 22946.719,E2 22946.719} C_VEL
LIN {X 0,Y 471.934,Z 848.456,A -85,B 0,C 180,E1 22944.162,E2 22944.162} C_VEL
LIN {X 0,Y 472.014,Z 843.904,A -85,B 0,C 180,E1 22941.472,E2 22941.472} C_VEL
LIN {X 0,Y 472.193,Z 838.246,A -85,B 0,C 180,E1 22939.013,E2 22939.013} C_VEL
LIN {X 0,Y 472.526,Z 830.877,A -85,B 0,C 180,E1 22936.539,E2 22936.539} C_VEL
LIN {X 0,Y 473.12,Z 821.347,A -85,B 0,C 180,E1 22933.927,E2 22933.927} C_VEL
LIN {X 0,Y 473.975,Z 810.346,A -85,B 0,C 180,E1 22931.425,E2 22931.425} C_VEL
LIN {X 0,Y 475.083,Z 797.751,A -85,B 0,C 180,E1 22929.035,E2 22929.035} C_VEL
LIN {X 0,Y 476.474,Z 783.702,A -85,B 0,C 180,E1 22926.764,E2 22926.764} C_VEL
LIN {X 0,Y 478.089,Z 768.7,A -85,B 0,C 180,E1 22924.678,E2 22924.678} C_VEL
LIN {X 0,Y 479.924,Z 752.231,A -85,B 0,C 180,E1 22922.719,E2 22922.719} C_VEL
LIN {X 0,Y 481.487,Z 737.1,A -85,B 0,C 180,E1 22921.198,E2 22921.198} C_VEL
LIN {X 0,Y 483.228,Z 718.362,A -85,B 0,C 180,E1 22919.636,E2 22919.636} C_VEL
LIN {X 0,Y 484.932,Z 697.908,A -85,B 0,C 180,E1 22918.209,E2 22918.209} C_VEL
LIN {X 0,Y 486.556,Z 677.003,A -85,B 0,C 180,E1 22917.004,E2 22917.004} C_VEL
LIN {X 0,Y 488.014,Z 655.408,A -85,B 0,C 180,E1 22915.99,E2 22915.99} C_VEL
LIN {X 0,Y 489.308,Z 632.893,A -85,B 0,C 180,E1 22915.165,E2 22915.165} C_VEL
LIN {X 0,Y 490.297,Z 611.071,A -85,B 0,C 180,E1 22914.59,E2 22914.59} C_VEL
LIN {X 0,Y 490.974,Z 581.066,A -85,B 0,C 180,E1 22914.058,E2 22914.058} C_VEL
LIN {X 0,Y 493.584,Z 430.546,A -85,B 0,C 180,E1 22911.619,E2 22911.619} C_VEL
LIN {X 0,Y 496.073,Z 327.503,A -85,B 0,C 180,E1 22909.787,E2 22909.787} C_VEL
LIN {X 0,Y 491.254,Z 296.385,A -85,B 0,C 180,E1 22908.614,E2 22908.614} C_VEL
LIN {X 0,Y 487.702,Z 289.972,A -85,B 0,C 180,E1 22908.06,E2 22908.06} C_VEL
LIN {X 0,Y 481.638,Z 273.393,A -85,B 0,C 180,E1 22905.913,E2 22905.913} C_VEL
LIN {X 0,Y 476.907,Z 262.437,A -85,B 0,C 180,E1 22904.19,E2 22904.19} C_VEL
LIN {X 0,Y 474.728,Z 257.967,A -85,B 0,C 180,E1 22903.363,E2 22903.363} C_VEL
LIN {X 0,Y 472.988,Z 254.341,A -85,B 0,C 180,E1 22902.637,E2 22902.637} C_VEL
LIN {X 0,Y 472.899,Z 253.831,A -85,B 0,C 180,E1 22902.488,E2 22902.488} C_VEL
LIN {X 0,Y 472.954,Z 253.824,A -85,B 0,C 180,E1 22899.051,E2 22899.051} C_VEL
LIN {X 0,Y 472.912,Z 253.83,A -85,B 0,C 180,E1 22895.403,E2 22895.403} C_VEL
LIN {X 0,Y 472.882,Z 253.833,A -85,B 0,C 180,E1 22891.912,E2 22891.912} C_VEL
LIN {X 0,Y 472.924,Z 254.011,A -85,B 0,C 180,E1 22888.469,E2 22888.469} C_VEL
LIN {X 0,Y 474.124,Z 257.22,A -85,B 0,C 180,E1 22888.175,E2 22888.175} C_VEL
LIN {X 0,Y 476.876,Z 260.202,A -85,B 0,C 180,E1 22887.675,E2 22887.675} C_VEL
LIN {X 0,Y 479.489,Z 264.156,A -85,B 0,C 180,E1 22887.193,E2 22887.193} C_VEL
LIN {X 0,Y 486.263,Z 274.296,A -85,B 0,C 180,E1 22886.063,E2 22886.063} C_VEL
LIN {X 0,Y 495.94,Z 290.404,A -85,B 0,C 180,E1 22884.639,E2 22884.639} C_VEL
LIN {X 0,Y 496.338,Z 291.663,A -85,B 0,C 180,E1 22884.571,E2 22884.571} C_VEL
LIN {X 0,Y 493.016,Z 417.507,A -85,B 0,C 180,E1 22882.36,E2 22882.36} C_VEL
LIN {X 0,Y 490.832,Z 533.669,A -85,B 0,C 180,E1 22880.443,E2 22880.443} C_VEL
LIN {X 0,Y 489.924,Z 555.274,A -85,B 0,C 180,E1 22879.878,E2 22879.878} C_VEL
LIN {X 0,Y 488.754,Z 576.5,A -85,B 0,C 180,E1 22879.107,E2 22879.107} C_VEL
LIN {X 0,Y 487.369,Z 596.593,A -85,B 0,C 180,E1 22878.171,E2 22878.171} C_VEL
LIN {X 0,Y 485.657,Z 616.694,A -85,B 0,C 180,E1 22877,E2 22877} C_VEL
LIN {X 0,Y 483.89,Z 635.556,A -85,B 0,C 180,E1 22875.656,E2 22875.656} C_VEL
LIN {X 0,Y 481.897,Z 654.413,A -85,B 0,C 180,E1 22874.051,E2 22874.051} C_VEL
LIN {X 0,Y 479.893,Z 672.455,A -85,B 0,C 180,E1 22872.21,E2 22872.21} C_VEL
LIN {X 0,Y 478.068,Z 689.015,A -85,B 0,C 180,E1 22870.242,E2 22870.242} C_VEL
LIN {X 0,Y 476.331,Z 705.253,A -85,B 0,C 180,E1 22867.965,E2 22867.965} C_VEL
LIN {X 0,Y 474.96,Z 719.136,A -85,B 0,C 180,E1 22865.68,E2 22865.68} C_VEL
LIN {X 0,Y 473.822,Z 732.167,A -85,B 0,C 180,E1 22863.147,E2 22863.147} C_VEL
LIN {X 0,Y 473.013,Z 743.045,A -85,B 0,C 180,E1 22860.607,E2 22860.607} C_VEL
LIN {X 0,Y 472.462,Z 752.474,A -85,B 0,C 180,E1 22857.94,E2 22857.94} C_VEL
LIN {X 0,Y 472.139,Z 759.944,A -85,B 0,C 180,E1 22855.264,E2 22855.264} C_VEL
LIN {X 0,Y 471.986,Z 765.472,A -85,B 0,C 180,E1 22852.7,E2 22852.7} C_VEL
LIN {X 0,Y 471.917,Z 769.363,A -85,B 0,C 180,E1 22850.12,E2 22850.12} C_VEL
LIN {X 0,Y 471.907,Z 771.786,A -85,B 0,C 180,E1 22847.397,E2 22847.397} C_VEL
LIN {X 0,Y 471.908,Z 772.479,A -85,B 0,C 180,E1 22844.77,E2 22844.77} C_VEL
LIN {X 0,Y 471.909,Z 771.529,A -85,B 0,C 180,E1 22842.11,E2 22842.11} C_VEL
LIN {X 0,Y 471.925,Z 768.967,A -85,B 0,C 180,E1 22839.466,E2 22839.466} C_VEL
LIN {X 0,Y 472.003,Z 764.676,A -85,B 0,C 180,E1 22836.798,E2 22836.798} C_VEL
LIN {X 0,Y 472.177,Z 758.69,A -85,B 0,C 180,E1 22834.14,E2 22834.14} C_VEL
LIN {X 0,Y 472.521,Z 751.17,A -85,B 0,C 180,E1 22831.571,E2 22831.571} C_VEL
LIN {X 0,Y 473.137,Z 741.301,A -85,B 0,C 180,E1 22828.857,E2 22828.857} C_VEL
LIN {X 0,Y 474.001,Z 729.968,A -85,B 0,C 180,E1 22826.308,E2 22826.308} C_VEL
LIN {X 0,Y 475.14,Z 717.295,A -85,B 0,C 180,E1 22823.902,E2 22823.902} C_VEL
LIN {X 0,Y 476.555,Z 703.022,A -85,B 0,C 180,E1 22821.611,E2 22821.611} C_VEL
LIN {X 0,Y 478.252,Z 687.277,A -85,B 0,C 180,E1 22819.447,E2 22819.447} C_VEL
LIN {X 0,Y 480.263,Z 669.109,A -85,B 0,C 180,E1 22817.335,E2 22817.335} C_VEL
LIN {X 0,Y 482.215,Z 651.469,A -85,B 0,C 180,E1 22815.593,E2 22815.593} C_VEL
LIN {X 0,Y 484.257,Z 632.041,A -85,B 0,C 180,E1 22813.977,E2 22813.977} C_VEL
LIN {X 0,Y 486.217,Z 611.639,A -85,B 0,C 180,E1 22812.576,E2 22812.576} C_VEL
LIN {X 0,Y 487.963,Z 590.996,A -85,B 0,C 180,E1 22811.418,E2 22811.418} C_VEL
LIN {X 0,Y 489.513,Z 569.127,A -85,B 0,C 180,E1 22810.448,E2 22810.448} C_VEL
LIN {X 0,Y 490.718,Z 547.668,A -85,B 0,C 180,E1 22809.727,E2 22809.727} C_VEL
LIN {X 0,Y 491.607,Z 524.81,A -85,B 0,C 180,E1 22809.194,E2 22809.194} C_VEL
LIN {X 0,Y 492.087,Z 500.873,A -85,B 0,C 180,E1 22808.801,E2 22808.801} C_VEL
LIN {X 0,Y 491.409,Z 493.306,A -85,B 0,C 180,E1 22808.614,E2 22808.614} C_VEL
LIN {X 0,Y 486.679,Z 473.598,A -85,B 0,C 180,E1 22807.865,E2 22807.865} C_VEL
LIN {X 0,Y 486.203,Z 467.096,A -85,B 0,C 180,E1 22807.705,E2 22807.705} C_VEL
LIN {X 0,Y 490.178,Z 294.151,A -85,B 0,C 180,E1 22804.76,E2 22804.76} C_VEL
LIN {X 0,Y 476.956,Z 273.625,A -85,B 0,C 180,E1 22802.975,E2 22802.975} C_VEL
LIN {X 0,Y 470.422,Z 264.08,A -85,B 0,C 180,E1 22802.045,E2 22802.045} C_VEL
LIN {X 0,Y 467.619,Z 259.796,A -85,B 0,C 180,E1 22801.628,E2 22801.628} C_VEL
LIN {X 0,Y 465.527,Z 256.792,A -85,B 0,C 180,E1 22801.318,E2 22801.318} C_VEL
LIN {X 0,Y 465.019,Z 254.814,A -85,B 0,C 180,E1 22801.212,E2 22801.212} C_VEL
LIN {X 0,Y 465.007,Z 254.813,A -85,B 0,C 180,E1 22797.536,E2 22797.536} C_VEL
LIN {X 0,Y 464.979,Z 254.815,A -85,B 0,C 180,E1 22793.959,E2 22793.959} C_VEL
LIN {X 0,Y 464.977,Z 254.816,A -85,B 0,C 180,E1 22790.256,E2 22790.256} C_VEL
LIN {X 0,Y 464.997,Z 254.811,A -85,B 0,C 180,E1 22786.619,E2 22786.619} C_VEL
LIN {X 0,Y 465.017,Z 254.808,A -85,B 0,C 180,E1 22783.049,E2 22783.049} C_VEL
LIN {X 0,Y 464.99,Z 254.812,A -85,B 0,C 180,E1 22779.407,E2 22779.407} C_VEL
LIN {X 0,Y 464.969,Z 254.809,A -85,B 0,C 180,E1 22775.802,E2 22775.802} C_VEL
LIN {X 0,Y 464.972,Z 254.81,A -85,B 0,C 180,E1 22772.096,E2 22772.096} C_VEL
LIN {X 0,Y 465.003,Z 254.807,A -85,B 0,C 180,E1 22768.523,E2 22768.523} C_VEL
LIN {X 0,Y 465.011,Z 254.803,A -85,B 0,C 180,E1 22764.82,E2 22764.82} C_VEL
LIN {X 0,Y 464.971,Z 254.807,A -85,B 0,C 180,E1 22761.344,E2 22761.344} C_VEL
LIN {X 0,Y 464.963,Z 254.811,A -85,B 0,C 180,E1 22757.71,E2 22757.71} C_VEL
LIN {X 0,Y 464.985,Z 254.81,A -85,B 0,C 180,E1 22754.153,E2 22754.153} C_VEL
LIN {X 0,Y 465.012,Z 254.807,A -85,B 0,C 180,E1 22750.534,E2 22750.534} C_VEL
LIN {X 0,Y 464.977,Z 254.812,A -85,B 0,C 180,E1 22746.962,E2 22746.962} C_VEL
LIN {X 0,Y 464.958,Z 254.815,A -85,B 0,C 180,E1 22743.432,E2 22743.432} C_VEL
LIN {X 0,Y 464.97,Z 254.817,A -85,B 0,C 180,E1 22739.814,E2 22739.814} C_VEL
LIN {X 0,Y 465.005,Z 254.81,A -85,B 0,C 180,E1 22736.308,E2 22736.308} C_VEL
LIN {X 0,Y 464.978,Z 254.809,A -85,B 0,C 180,E1 22732.673,E2 22732.673} C_VEL
LIN {X 0,Y 464.951,Z 254.814,A -85,B 0,C 180,E1 22729.178,E2 22729.178} C_VEL
LIN {X 0,Y 464.962,Z 254.817,A -85,B 0,C 180,E1 22725.552,E2 22725.552} C_VEL
LIN {X 0,Y 464.997,Z 254.819,A -85,B 0,C 180,E1 22721.931,E2 22721.931} C_VEL
LIN {X 0,Y 464.989,Z 254.81,A -85,B 0,C 180,E1 22718.296,E2 22718.296} C_VEL
LIN {X 0,Y 464.95,Z 254.81,A -85,B 0,C 180,E1 22714.738,E2 22714.738} C_VEL
LIN {X 0,Y 464.945,Z 254.813,A -85,B 0,C 180,E1 22711.069,E2 22711.069} C_VEL
LIN {X 0,Y 464.98,Z 254.816,A -85,B 0,C 180,E1 22707.638,E2 22707.638} C_VEL
LIN {X 0,Y 464.994,Z 254.813,A -85,B 0,C 180,E1 22703.96,E2 22703.96} C_VEL
LIN {X 0,Y 464.946,Z 254.814,A -85,B 0,C 180,E1 22700.517,E2 22700.517} C_VEL
LIN {X 0,Y 464.939,Z 254.816,A -85,B 0,C 180,E1 22696.874,E2 22696.874} C_VEL
LIN {X 0,Y 464.974,Z 254.817,A -85,B 0,C 180,E1 22693.427,E2 22693.427} C_VEL
LIN {X 0,Y 464.985,Z 254.813,A -85,B 0,C 180,E1 22689.779,E2 22689.779} C_VEL
LIN {X 0,Y 464.938,Z 254.816,A -85,B 0,C 180,E1 22686.295,E2 22686.295} C_VEL
LIN {X 0,Y 464.934,Z 254.818,A -85,B 0,C 180,E1 22682.71,E2 22682.71} C_VEL
LIN {X 0,Y 464.967,Z 254.818,A -85,B 0,C 180,E1 22679.17,E2 22679.17} C_VEL
LIN {X 0,Y 464.987,Z 254.818,A -85,B 0,C 180,E1 22675.559,E2 22675.559} C_VEL
LIN {X 0,Y 464.944,Z 254.817,A -85,B 0,C 180,E1 22672.088,E2 22672.088} C_VEL
LIN {X 0,Y 464.939,Z 254.815,A -85,B 0,C 180,E1 22668.462,E2 22668.462} C_VEL
LIN {X 0,Y 464.968,Z 254.816,A -85,B 0,C 180,E1 22664.903,E2 22664.903} C_VEL
LIN {X 0,Y 464.995,Z 254.811,A -85,B 0,C 180,E1 22661.312,E2 22661.312} C_VEL
LIN {X 0,Y 464.956,Z 254.815,A -85,B 0,C 180,E1 22657.759,E2 22657.759} C_VEL
LIN {X 0,Y 464.945,Z 254.814,A -85,B 0,C 180,E1 22654.252,E2 22654.252} C_VEL
LIN {X 0,Y 464.983,Z 254.812,A -85,B 0,C 180,E1 22650.782,E2 22650.782} C_VEL
LIN {X 0,Y 464.996,Z 254.814,A -85,B 0,C 180,E1 22647.188,E2 22647.188} C_VEL
LIN {X 0,Y 464.954,Z 254.818,A -85,B 0,C 180,E1 22643.744,E2 22643.744} C_VEL
LIN {X 0,Y 464.955,Z 254.819,A -85,B 0,C 180,E1 22640.145,E2 22640.145} C_VEL
LIN {X 0,Y 464.994,Z 254.97,A -85,B 0,C 180,E1 22638.457,E2 22638.457} C_VEL
LIN {X 0,Y 466.162,Z 258.156,A -85,B 0,C 180,E1 22637.994,E2 22637.994} C_VEL
LIN {X 0,Y 467.316,Z 260.443,A -85,B 0,C 180,E1 22637.625,E2 22637.625} C_VEL
LIN {X 0,Y 474.444,Z 275.483,A -85,B 0,C 180,E1 22635.345,E2 22635.345} C_VEL
LIN {X 0,Y 482.307,Z 293.577,A -85,B 0,C 180,E1 22632.839,E2 22632.839} C_VEL
LIN {X 0,Y 484.77,Z 299.43,A -85,B 0,C 180,E1 22632.119,E2 22632.119} C_VEL
LIN {X 0,Y 486.277,Z 302.467,A -85,B 0,C 180,E1 22631.898,E2 22631.898} C_VEL
LIN {X 0,Y 490.792,Z 331.229,A -85,B 0,C 180,E1 22630.843,E2 22630.843} C_VEL
LIN {X 0,Y 486.095,Z 536.473,A -85,B 0,C 180,E1 22627.374,E2 22627.374} C_VEL
LIN {X 0,Y 484.467,Z 608.157,A -85,B 0,C 180,E1 22626.15,E2 22626.15} C_VEL
LIN {X 0,Y 483.359,Z 629.788,A -85,B 0,C 180,E1 22625.581,E2 22625.581} C_VEL
LIN {X 0,Y 481.918,Z 651.707,A -85,B 0,C 180,E1 22624.787,E2 22624.787} C_VEL
LIN {X 0,Y 480.235,Z 673.414,A -85,B 0,C 180,E1 22623.771,E2 22623.771} C_VEL
LIN {X 0,Y 478.477,Z 693.18,A -85,B 0,C 180,E1 22622.623,E2 22622.623} C_VEL
LIN {X 0,Y 476.515,Z 713.228,A -85,B 0,C 180,E1 22621.215,E2 22621.215} C_VEL
LIN {X 0,Y 474.443,Z 733.201,A -85,B 0,C 180,E1 22619.545,E2 22619.545} C_VEL
LIN {X 0,Y 472.595,Z 750.744,A -85,B 0,C 180,E1 22617.827,E2 22617.827} C_VEL
LIN {X 0,Y 470.743,Z 767.645,A -85,B 0,C 180,E1 22615.878,E2 22615.878} C_VEL
LIN {X 0,Y 469,Z 782.872,A -85,B 0,C 180,E1 22613.76,E2 22613.76} C_VEL
LIN {X 0,Y 467.505,Z 796.738,A -85,B 0,C 180,E1 22611.511,E2 22611.511} C_VEL
LIN {X 0,Y 466.286,Z 809.09,A -85,B 0,C 180,E1 22609.151,E2 22609.151} C_VEL
LIN {X 0,Y 465.357,Z 819.813,A -85,B 0,C 180,E1 22606.731,E2 22606.731} C_VEL
LIN {X 0,Y 464.7,Z 829.266,A -85,B 0,C 180,E1 22604.197,E2 22604.197} C_VEL
LIN {X 0,Y 464.287,Z 836.884,A -85,B 0,C 180,E1 22601.678,E2 22601.678} C_VEL
LIN {X 0,Y 464.046,Z 843.148,A -85,B 0,C 180,E1 22599.048,E2 22599.048} C_VEL
LIN {X 0,Y 463.946,Z 847.685,A -85,B 0,C 180,E1 22596.529,E2 22596.529} C_VEL
LIN {X 0,Y 463.91,Z 850.674,A -85,B 0,C 180,E1 22593.954,E2 22593.954} C_VEL
LIN {X 0,Y 463.903,Z 852.258,A -85,B 0,C 180,E1 22591.357,E2 22591.357} C_VEL
LIN {X 0,Y 463.911,Z 852.303,A -85,B 0,C 180,E1 22588.887,E2 22588.887} C_VEL
LIN {X 0,Y 463.91,Z 850.782,A -85,B 0,C 180,E1 22586.168,E2 22586.168} C_VEL
LIN {X 0,Y 463.942,Z 847.816,A -85,B 0,C 180,E1 22583.564,E2 22583.564} C_VEL
LIN {X 0,Y 464.034,Z 843.396,A -85,B 0,C 180,E1 22581.074,E2 22581.074} C_VEL
LIN {X 0,Y 464.272,Z 837.23,A -85,B 0,C 180,E1 22578.445,E2 22578.445} C_VEL
LIN {X 0,Y 464.673,Z 829.661,A -85,B 0,C 180,E1 22575.927,E2 22575.927} C_VEL
LIN {X 0,Y 465.32,Z 820.316,A -85,B 0,C 180,E1 22573.393,E2 22573.393} C_VEL
LIN {X 0,Y 466.233,Z 809.713,A -85,B 0,C 180,E1 22570.975,E2 22570.975} C_VEL
LIN {X 0,Y 467.389,Z 797.75,A -85,B 0,C 180,E1 22568.673,E2 22568.673} C_VEL
LIN {X 0,Y 468.903,Z 783.7,A -85,B 0,C 180,E1 22566.366,E2 22566.366} C_VEL
LIN {X 0,Y 470.623,Z 768.797,A -85,B 0,C 180,E1 22564.265,E2 22564.265} C_VEL
LIN {X 0,Y 472.047,Z 755.012,A -85,B 0,C 180,E1 22562.67,E2 22562.67} C_VEL
LIN {X 0,Y 473.903,Z 736.46,A -85,B 0,C 180,E1 22560.831,E2 22560.831} C_VEL
LIN {X 0,Y 475.771,Z 717.44,A -85,B 0,C 180,E1 22559.227,E2 22559.227} C_VEL
LIN {X 0,Y 477.542,Z 697.223,A -85,B 0,C 180,E1 22557.8,E2 22557.8} C_VEL
LIN {X 0,Y 479.308,Z 675.917,A -85,B 0,C 180,E1 22556.556,E2 22556.556} C_VEL
LIN {X 0,Y 480.857,Z 654.087,A -85,B 0,C 180,E1 22555.521,E2 22555.521} C_VEL
LIN {X 0,Y 482.265,Z 631.406,A -85,B 0,C 180,E1 22554.686,E2 22554.686} C_VEL
LIN {X 0,Y 483.322,Z 609.08,A -85,B 0,C 180,E1 22554.096,E2 22554.096} C_VEL
LIN {X 0,Y 484.063,Z 577.376,A -85,B 0,C 180,E1 22553.534,E2 22553.534} C_VEL
LIN {X 0,Y 486.705,Z 441.558,A -85,B 0,C 180,E1 22551.281,E2 22551.281} C_VEL
LIN {X 0,Y 489.956,Z 329.692,A -85,B 0,C 180,E1 22549.244,E2 22549.244} C_VEL
LIN {X 0,Y 485.704,Z 300.608,A -85,B 0,C 180,E1 22548.111,E2 22548.111} C_VEL
LIN {X 0,Y 478.696,Z 286.934,A -85,B 0,C 180,E1 22546.888,E2 22546.888} C_VEL
LIN {X 0,Y 474.067,Z 274.58,A -85,B 0,C 180,E1 22545.127,E2 22545.127} C_VEL
LIN {X 0,Y 470.326,Z 266.386,A -85,B 0,C 180,E1 22543.703,E2 22543.703} C_VEL
LIN {X 0,Y 468.766,Z 262.968,A -85,B 0,C 180,E1 22543.044,E2 22543.044} C_VEL
LIN {X 0,Y 466.983,Z 259.226,A -85,B 0,C 180,E1 22542.246,E2 22542.246} C_VEL
LIN {X 0,Y 465.173,Z 255.811,A -85,B 0,C 180,E1 22541.396,E2 22541.396} C_VEL
LIN {X 0,Y 465.009,Z 254.815,A -85,B 0,C 180,E1 22541.145,E2 22541.145} C_VEL
LIN {X 0,Y 464.958,Z 254.819,A -85,B 0,C 180,E1 22537.643,E2 22537.643} C_VEL
LIN {X 0,Y 464.945,Z 254.821,A -85,B 0,C 180,E1 22533.996,E2 22533.996} C_VEL
LIN {X 0,Y 464.951,Z 254.821,A -85,B 0,C 180,E1 22530.356,E2 22530.356} C_VEL
LIN {X 0,Y 464.973,Z 255.044,A -85,B 0,C 180,E1 22529.836,E2 22529.836} C_VEL
LIN {X 0,Y 466.177,Z 258.172,A -85,B 0,C 180,E1 22529.483,E2 22529.483} C_VEL
LIN {X 0,Y 469.218,Z 261.312,A -85,B 0,C 180,E1 22528.824,E2 22528.824} C_VEL
LIN {X 0,Y 471.58,Z 265.15,A -85,B 0,C 180,E1 22528.305,E2 22528.305} C_VEL
LIN {X 0,Y 473.202,Z 267.088,A -85,B 0,C 180,E1 22527.998,E2 22527.998} C_VEL
LIN {X 0,Y 477.225,Z 273.203,A -85,B 0,C 180,E1 22527.235,E2 22527.235} C_VEL
LIN {X 0,Y 482.346,Z 281.082,A -85,B 0,C 180,E1 22526.355,E2 22526.355} C_VEL
LIN {X 0,Y 490.216,Z 294.402,A -85,B 0,C 180,E1 22525.136,E2 22525.136} C_VEL
LIN {X 0,Y 486.691,Z 407.298,A -85,B 0,C 180,E1 22523.078,E2 22523.078} C_VEL
LIN {X 0,Y 483.923,Z 535.316,A -85,B 0,C 180,E1 22520.897,E2 22520.897} C_VEL
LIN {X 0,Y 482.981,Z 556.961,A -85,B 0,C 180,E1 22520.318,E2 22520.318} C_VEL
LIN {X 0,Y 481.807,Z 577.431,A -85,B 0,C 180,E1 22519.563,E2 22519.563} C_VEL
LIN {X 0,Y 480.398,Z 597.25,A -85,B 0,C 180,E1 22518.633,E2 22518.633} C_VEL
LIN {X 0,Y 478.694,Z 616.497,A -85,B 0,C 180,E1 22517.505,E2 22517.505} C_VEL
LIN {X 0,Y 476.815,Z 635.731,A -85,B 0,C 180,E1 22516.133,E2 22516.133} C_VEL
LIN {X 0,Y 474.74,Z 654.646,A -85,B 0,C 180,E1 22514.516,E2 22514.516} C_VEL
LIN {X 0,Y 472.739,Z 671.747,A -85,B 0,C 180,E1 22512.77,E2 22512.77} C_VEL
LIN {X 0,Y 470.721,Z 688.282,A -85,B 0,C 180,E1 22510.775,E2 22510.775} C_VEL
LIN {X 0,Y 468.729,Z 705.369,A -85,B 0,C 180,E1 22508.342,E2 22508.342} C_VEL
LIN {X 0,Y 467.245,Z 719.229,A -85,B 0,C 180,E1 22506.02,E2 22506.02} C_VEL
LIN {X 0,Y 466.006,Z 732.245,A -85,B 0,C 180,E1 22503.446,E2 22503.446} C_VEL
LIN {X 0,Y 465.121,Z 743.103,A -85,B 0,C 180,E1 22500.864,E2 22500.864} C_VEL
LIN {X 0,Y 464.519,Z 752.522,A -85,B 0,C 180,E1 22498.151,E2 22498.151} C_VEL
LIN {X 0,Y 464.165,Z 759.977,A -85,B 0,C 180,E1 22495.43,E2 22495.43} C_VEL
LIN {X 0,Y 463.995,Z 765.493,A -85,B 0,C 180,E1 22492.822,E2 22492.822} C_VEL
LIN {X 0,Y 463.921,Z 769.374,A -85,B 0,C 180,E1 22490.199,E2 22490.199} C_VEL
LIN {X 0,Y 463.906,Z 771.792,A -85,B 0,C 180,E1 22487.429,E2 22487.429} C_VEL
LIN {X 0,Y 463.911,Z 772.494,A -85,B 0,C 180,E1 22484.885,E2 22484.885} C_VEL
LIN {X 0,Y 463.909,Z 771.604,A -85,B 0,C 180,E1 22482.181,E2 22482.181} C_VEL
LIN {X 0,Y 463.928,Z 769.052,A -85,B 0,C 180,E1 22479.436,E2 22479.436} C_VEL
LIN {X 0,Y 464.008,Z 764.907,A -85,B 0,C 180,E1 22476.778,E2 22476.778} C_VEL
LIN {X 0,Y 464.194,Z 758.989,A -85,B 0,C 180,E1 22474.074,E2 22474.074} C_VEL
LIN {X 0,Y 464.574,Z 751.42,A -85,B 0,C 180,E1 22471.415,E2 22471.415} C_VEL
LIN {X 0,Y 465.234,Z 741.638,A -85,B 0,C 180,E1 22468.664,E2 22468.664} C_VEL
LIN {X 0,Y 466.154,Z 730.555,A -85,B 0,C 180,E1 22466.108,E2 22466.108} C_VEL
LIN {X 0,Y 467.456,Z 717.294,A -85,B 0,C 180,E1 22463.538,E2 22463.538} C_VEL
LIN {X 0,Y 469.009,Z 702.888,A -85,B 0,C 180,E1 22461.191,E2 22461.191} C_VEL
LIN {X 0,Y 470.848,Z 687.164,A -85,B 0,C 180,E1 22458.995,E2 22458.995} C_VEL
LIN {X 0,Y 472.939,Z 669.822,A -85,B 0,C 180,E1 22456.935,E2 22456.935} C_VEL
LIN {X 0,Y 475.026,Z 652.126,A -85,B 0,C 180,E1 22455.164,E2 22455.164} C_VEL
LIN {X 0,Y 477.087,Z 633.5,A -85,B 0,C 180,E1 22453.592,E2 22453.592} C_VEL
LIN {X 0,Y 479.11,Z 613.734,A -85,B 0,C 180,E1 22452.2,E2 22452.2} C_VEL
LIN {X 0,Y 480.882,Z 594.369,A -85,B 0,C 180,E1 22451.075,E2 22451.075} C_VEL
LIN {X 0,Y 482.498,Z 573.012,A -85,B 0,C 180,E1 22450.081,E2 22450.081} C_VEL
LIN {X 0,Y 483.841,Z 551.226,A -85,B 0,C 180,E1 22449.31,E2 22449.31} C_VEL
LIN {X 0,Y 484.84,Z 529.062,A -85,B 0,C 180,E1 22448.749,E2 22448.749} C_VEL
LIN {X 0,Y 486.203,Z 467.096,A -85,B 0,C 180,E1 22447.705,E2 22447.705} C_VEL
LIN {X 0,Y 485.556,Z 459.535,A -85,B 0,C 180,E1 22447.509,E2 22447.509} C_VEL
LIN {X 0,Y 480.95,Z 439.839,A -85,B 0,C 180,E1 22446.737,E2 22446.737} C_VEL
LIN {X 0,Y 480.507,Z 433.338,A -85,B 0,C 180,E1 22446.573,E2 22446.573} C_VEL
LIN {X 0,Y 483.97,Z 297.508,A -85,B 0,C 180,E1 22444.211,E2 22444.211} C_VEL
LIN {X 0,Y 471.68,Z 278.452,A -85,B 0,C 180,E1 22442.505,E2 22442.505} C_VEL
LIN {X 0,Y 462.786,Z 265.377,A -85,B 0,C 180,E1 22441.198,E2 22441.198} C_VEL
LIN {X 0,Y 459.756,Z 260.861,A -85,B 0,C 180,E1 22440.736,E2 22440.736} C_VEL
LIN {X 0,Y 457.592,Z 257.886,A -85,B 0,C 180,E1 22440.406,E2 22440.406} C_VEL
LIN {X 0,Y 457.04,Z 255.806,A -85,B 0,C 180,E1 22440.276,E2 22440.276} C_VEL
LIN {X 0,Y 457.054,Z 255.802,A -85,B 0,C 180,E1 22436.646,E2 22436.646} C_VEL
LIN {X 0,Y 457.076,Z 255.798,A -85,B 0,C 180,E1 22432.917,E2 22432.917} C_VEL
LIN {X 0,Y 457.072,Z 255.801,A -85,B 0,C 180,E1 22429.289,E2 22429.289} C_VEL
LIN {X 0,Y 457.046,Z 255.8,A -85,B 0,C 180,E1 22425.611,E2 22425.611} C_VEL
LIN {X 0,Y 457.034,Z 255.802,A -85,B 0,C 180,E1 22421.996,E2 22421.996} C_VEL
LIN {X 0,Y 457.041,Z 255.8,A -85,B 0,C 180,E1 22418.303,E2 22418.303} C_VEL
LIN {X 0,Y 457.073,Z 255.796,A -85,B 0,C 180,E1 22414.769,E2 22414.769} C_VEL
LIN {X 0,Y 457.07,Z 255.796,A -85,B 0,C 180,E1 22411.004,E2 22411.004} C_VEL
LIN {X 0,Y 457.037,Z 255.799,A -85,B 0,C 180,E1 22407.368,E2 22407.368} C_VEL
LIN {X 0,Y 457.026,Z 255.801,A -85,B 0,C 180,E1 22403.721,E2 22403.721} C_VEL
LIN {X 0,Y 457.036,Z 255.802,A -85,B 0,C 180,E1 22400.049,E2 22400.049} C_VEL
LIN {X 0,Y 457.074,Z 255.801,A -85,B 0,C 180,E1 22396.465,E2 22396.465} C_VEL
LIN {X 0,Y 457.058,Z 255.799,A -85,B 0,C 180,E1 22392.824,E2 22392.824} C_VEL
LIN {X 0,Y 457.026,Z 255.8,A -85,B 0,C 180,E1 22389.244,E2 22389.244} C_VEL
LIN {X 0,Y 457.02,Z 255.8,A -85,B 0,C 180,E1 22385.514,E2 22385.514} C_VEL
LIN {X 0,Y 457.041,Z 255.799,A -85,B 0,C 180,E1 22381.945,E2 22381.945} C_VEL
LIN {X 0,Y 457.07,Z 255.8,A -85,B 0,C 180,E1 22378.333,E2 22378.333} C_VEL
LIN {X 0,Y 457.042,Z 255.805,A -85,B 0,C 180,E1 22374.682,E2 22374.682} C_VEL
LIN {X 0,Y 457.015,Z 255.806,A -85,B 0,C 180,E1 22371.107,E2 22371.107} C_VEL
LIN {X 0,Y 457.018,Z 255.806,A -85,B 0,C 180,E1 22367.468,E2 22367.468} C_VEL
LIN {X 0,Y 457.05,Z 255.8,A -85,B 0,C 180,E1 22363.903,E2 22363.903} C_VEL
LIN {X 0,Y 457.062,Z 255.803,A -85,B 0,C 180,E1 22360.232,E2 22360.232} C_VEL
LIN {X 0,Y 457.017,Z 255.806,A -85,B 0,C 180,E1 22356.671,E2 22356.671} C_VEL
LIN {X 0,Y 457.006,Z 255.806,A -85,B 0,C 180,E1 22353.006,E2 22353.006} C_VEL
LIN {X 0,Y 457.026,Z 255.804,A -85,B 0,C 180,E1 22349.461,E2 22349.461} C_VEL
LIN {X 0,Y 457.056,Z 255.797,A -85,B 0,C 180,E1 22345.943,E2 22345.943} C_VEL
LIN {X 0,Y 457.017,Z 255.805,A -85,B 0,C 180,E1 22342.373,E2 22342.373} C_VEL
LIN {X 0,Y 457,Z 255.805,A -85,B 0,C 180,E1 22338.759,E2 22338.759} C_VEL
LIN {X 0,Y 457.009,Z 255.804,A -85,B 0,C 180,E1 22335.089,E2 22335.089} C_VEL
LIN {X 0,Y 457.049,Z 255.803,A -85,B 0,C 180,E1 22331.609,E2 22331.609} C_VEL
LIN {X 0,Y 457.03,Z 255.807,A -85,B 0,C 180,E1 22327.92,E2 22327.92} C_VEL
LIN {X 0,Y 456.996,Z 255.806,A -85,B 0,C 180,E1 22324.39,E2 22324.39} C_VEL
LIN {X 0,Y 456.995,Z 255.802,A -85,B 0,C 180,E1 22320.625,E2 22320.625} C_VEL
LIN {X 0,Y 457.025,Z 255.806,A -85,B 0,C 180,E1 22317.114,E2 22317.114} C_VEL
LIN {X 0,Y 457.059,Z 255.802,A -85,B 0,C 180,E1 22313.467,E2 22313.467} C_VEL
LIN {X 0,Y 457.024,Z 255.807,A -85,B 0,C 180,E1 22309.791,E2 22309.791} C_VEL
LIN {X 0,Y 457.002,Z 255.803,A -85,B 0,C 180,E1 22306.202,E2 22306.202} C_VEL
LIN {X 0,Y 457.005,Z 255.805,A -85,B 0,C 180,E1 22302.426,E2 22302.426} C_VEL
LIN {X 0,Y 457.033,Z 255.801,A -85,B 0,C 180,E1 22298.839,E2 22298.839} C_VEL
LIN {X 0,Y 457.061,Z 255.801,A -85,B 0,C 180,E1 22295.205,E2 22295.205} C_VEL
LIN {X 0,Y 457.028,Z 255.804,A -85,B 0,C 180,E1 22291.575,E2 22291.575} C_VEL
LIN {X 0,Y 457.01,Z 255.807,A -85,B 0,C 180,E1 22288.03,E2 22288.03} C_VEL
LIN {X 0,Y 457.023,Z 255.807,A -85,B 0,C 180,E1 22284.411,E2 22284.411} C_VEL
LIN {X 0,Y 457.062,Z 255.801,A -85,B 0,C 180,E1 22280.786,E2 22280.786} C_VEL
LIN {X 0,Y 457.045,Z 255.873,A -85,B 0,C 180,E1 22279.372,E2 22279.372} C_VEL
LIN {X 0,Y 458.52,Z 259.497,A -85,B 0,C 180,E1 22278.81,E2 22278.81} C_VEL
LIN {X 0,Y 466.692,Z 276.568,A -85,B 0,C 180,E1 22276.125,E2 22276.125} C_VEL
LIN {X 0,Y 474.361,Z 294.192,A -85,B 0,C 180,E1 22273.611,E2 22273.611} C_VEL
LIN {X 0,Y 476.381,Z 298.726,A -85,B 0,C 180,E1 22273.035,E2 22273.035} C_VEL
LIN {X 0,Y 480.631,Z 306.493,A -85,B 0,C 180,E1 22272.406,E2 22272.406} C_VEL
LIN {X 0,Y 484.65,Z 332.723,A -85,B 0,C 180,E1 22271.429,E2 22271.429} C_VEL
LIN {X 0,Y 479.619,Z 532.782,A -85,B 0,C 180,E1 22267.983,E2 22267.983} C_VEL
LIN {X 0,Y 477.782,Z 607.525,A -85,B 0,C 180,E1 22266.687,E2 22266.687} C_VEL
LIN {X 0,Y 476.584,Z 629.412,A -85,B 0,C 180,E1 22266.103,E2 22266.103} C_VEL
LIN {X 0,Y 475.001,Z 651.949,A -85,B 0,C 180,E1 22265.272,E2 22265.272} C_VEL
LIN {X 0,Y 473.129,Z 674.244,A -85,B 0,C 180,E1 22264.202,E2 22264.202} C_VEL
LIN {X 0,Y 471.177,Z 694.832,A -85,B 0,C 180,E1 22262.975,E2 22262.975} C_VEL
LIN {X 0,Y 469.099,Z 714.551,A -85,B 0,C 180,E1 22261.543,E2 22261.543} C_VEL
LIN {X 0,Y 466.918,Z 734.121,A -85,B 0,C 180,E1 22259.857,E2 22259.857} C_VEL
LIN {X 0,Y 464.869,Z 752.214,A -85,B 0,C 180,E1 22258.023,E2 22258.023} C_VEL
LIN {X 0,Y 462.945,Z 768.954,A -85,B 0,C 180,E1 22256.042,E2 22256.042} C_VEL
LIN {X 0,Y 461.212,Z 784.297,A -85,B 0,C 180,E1 22253.914,E2 22253.914} C_VEL
LIN {X 0,Y 459.881,Z 796.36,A -85,B 0,C 180,E1 22251.958,E2 22251.958} C_VEL
LIN {X 0,Y 458.57,Z 808.454,A -85,B 0,C 180,E1 22249.618,E2 22249.618} C_VEL
LIN {X 0,Y 457.499,Z 819.812,A -85,B 0,C 180,E1 22247.027,E2 22247.027} C_VEL
LIN {X 0,Y 456.779,Z 829.266,A -85,B 0,C 180,E1 22244.449,E2 22244.449} C_VEL
LIN {X 0,Y 456.327,Z 836.884,A -85,B 0,C 180,E1 22241.884,E2 22241.884} C_VEL
LIN {X 0,Y 456.069,Z 843.148,A -85,B 0,C 180,E1 22239.208,E2 22239.208} C_VEL
LIN {X 0,Y 455.948,Z 847.823,A -85,B 0,C 180,E1 22236.546,E2 22236.546} C_VEL
LIN {X 0,Y 455.91,Z 850.787,A -85,B 0,C 180,E1 22233.897,E2 22233.897} C_VEL
LIN {X 0,Y 455.911,Z 852.304,A -85,B 0,C 180,E1 22231.13,E2 22231.13} C_VEL
LIN {X 0,Y 455.904,Z 852.257,A -85,B 0,C 180,E1 22228.616,E2 22228.616} C_VEL
LIN {X 0,Y 455.912,Z 850.668,A -85,B 0,C 180,E1 22225.975,E2 22225.975} C_VEL
LIN {X 0,Y 455.953,Z 847.63,A -85,B 0,C 180,E1 22223.325,E2 22223.325} C_VEL
LIN {X 0,Y 456.069,Z 843.142,A -85,B 0,C 180,E1 22220.79,E2 22220.79} C_VEL
LIN {X 0,Y 456.341,Z 836.523,A -85,B 0,C 180,E1 22217.985,E2 22217.985} C_VEL
LIN {X 0,Y 456.83,Z 828.556,A -85,B 0,C 180,E1 22215.331,E2 22215.331} C_VEL
LIN {X 0,Y 457.594,Z 818.772,A -85,B 0,C 180,E1 22212.712,E2 22212.712} C_VEL
LIN {X 0,Y 458.631,Z 807.807,A -85,B 0,C 180,E1 22210.249,E2 22210.249} C_VEL
LIN {X 0,Y 459.965,Z 795.62,A -85,B 0,C 180,E1 22207.909,E2 22207.909} C_VEL
LIN {X 0,Y 461.209,Z 784.241,A -85,B 0,C 180,E1 22206.083,E2 22206.083} C_VEL
LIN {X 0,Y 462.871,Z 768.756,A -85,B 0,C 180,E1 22203.99,E2 22203.99} C_VEL
LIN {X 0,Y 464.702,Z 751.68,A -85,B 0,C 180,E1 22202.026,E2 22202.026} C_VEL
LIN {X 0,Y 466.657,Z 732.951,A -85,B 0,C 180,E1 22200.192,E2 22200.192} C_VEL
LIN {X 0,Y 468.719,Z 712.35,A -85,B 0,C 180,E1 22198.49,E2 22198.49} C_VEL
LIN {X 0,Y 470.573,Z 692.594,A -85,B 0,C 180,E1 22197.119,E2 22197.119} C_VEL
LIN {X 0,Y 472.295,Z 672.05,A -85,B 0,C 180,E1 22195.947,E2 22195.947} C_VEL
LIN {X 0,Y 473.911,Z 650.449,A -85,B 0,C 180,E1 22194.946,E2 22194.946} C_VEL
LIN {X 0,Y 475.321,Z 628.468,A -85,B 0,C 180,E1 22194.151,E2 22194.151} C_VEL
LIN {X 0,Y 476.438,Z 605.835,A -85,B 0,C 180,E1 22193.56,E2 22193.56} C_VEL
LIN {X 0,Y 477.365,Z 563.93,A -85,B 0,C 180,E1 22192.834,E2 22192.834} C_VEL
LIN {X 0,Y 480.221,Z 439.142,A -85,B 0,C 180,E1 22190.69,E2 22190.69} C_VEL
LIN {X 0,Y 483.821,Z 331.132,A -85,B 0,C 180,E1 22188.651,E2 22188.651} C_VEL
LIN {X 0,Y 480.181,Z 304.626,A -85,B 0,C 180,E1 22187.572,E2 22187.572} C_VEL
LIN {X 0,Y 471.528,Z 287.415,A -85,B 0,C 180,E1 22185.937,E2 22185.937} C_VEL
LIN {X 0,Y 469.476,Z 282.993,A -85,B 0,C 180,E1 22185.431,E2 22185.431} C_VEL
LIN {X 0,Y 465.42,Z 273.111,A -85,B 0,C 180,E1 22183.77,E2 22183.77} C_VEL
LIN {X 0,Y 461.856,Z 265.321,A -85,B 0,C 180,E1 22182.154,E2 22182.154} C_VEL
LIN {X 0,Y 459.891,Z 261.692,A -85,B 0,C 180,E1 22181.206,E2 22181.206} C_VEL
LIN {X 0,Y 459.459,Z 260.59,A -85,B 0,C 180,E1 22180.923,E2 22180.923} C_VEL
LIN {X 0,Y 457.422,Z 257.52,A -85,B 0,C 180,E1 22179.827,E2 22179.827} C_VEL
LIN {X 0,Y 457.052,Z 255.806,A -85,B 0,C 180,E1 22179.296,E2 22179.296} C_VEL
LIN {X 0,Y 457.013,Z 255.81,A -85,B 0,C 180,E1 22175.739,E2 22175.739} C_VEL
LIN {X 0,Y 457.005,Z 255.81,A -85,B 0,C 180,E1 22172.118,E2 22172.118} C_VEL
LIN {X 0,Y 457.037,Z 255.972,A -85,B 0,C 180,E1 22171.599,E2 22171.599} C_VEL
LIN {X 0,Y 458.174,Z 259.004,A -85,B 0,C 180,E1 22171.135,E2 22171.135} C_VEL
LIN {X 0,Y 461.015,Z 261.785,A -85,B 0,C 180,E1 22170.355,E2 22170.355} C_VEL
LIN {X 0,Y 461.751,Z 262.666,A -85,B 0,C 180,E1 22170.165,E2 22170.165} C_VEL
LIN {X 0,Y 464.048,Z 266.342,A -85,B 0,C 180,E1 22169.554,E2 22169.554} C_VEL
LIN {X 0,Y 465.743,Z 268.232,A -85,B 0,C 180,E1 22169.166,E2 22169.166} C_VEL
LIN {X 0,Y 468.757,Z 272.535,A -85,B 0,C 180,E1 22168.501,E2 22168.501} C_VEL
LIN {X 0,Y 475.326,Z 282.589,A -85,B 0,C 180,E1 22167.218,E2 22167.218} C_VEL
LIN {X 0,Y 483.499,Z 296.385,A -85,B 0,C 180,E1 22165.83,E2 22165.83} C_VEL
LIN {X 0,Y 484.178,Z 298.167,A -85,B 0,C 180,E1 22165.707,E2 22165.707} C_VEL
LIN {X 0,Y 480.375,Z 402.917,A -85,B 0,C 180,E1 22163.725,E2 22163.725} C_VEL
LIN {X 0,Y 477.047,Z 537.163,A -85,B 0,C 180,E1 22161.362,E2 22161.362} C_VEL
LIN {X 0,Y 476.062,Z 558.944,A -85,B 0,C 180,E1 22160.763,E2 22160.763} C_VEL
LIN {X 0,Y 474.81,Z 579.554,A -85,B 0,C 180,E1 22159.98,E2 22159.98} C_VEL
LIN {X 0,Y 473.254,Z 600.007,A -85,B 0,C 180,E1 22158.989,E2 22158.989} C_VEL
LIN {X 0,Y 471.419,Z 620.028,A -85,B 0,C 180,E1 22157.785,E2 22157.785} C_VEL
LIN {X 0,Y 469.462,Z 638.82,A -85,B 0,C 180,E1 22156.393,E2 22156.393} C_VEL
LIN {X 0,Y 467.292,Z 657.393,A -85,B 0,C 180,E1 22154.753,E2 22154.753} C_VEL
LIN {X 0,Y 465.229,Z 674.301,A -85,B 0,C 180,E1 22152.98,E2 22152.98} C_VEL
LIN {X 0,Y 463.126,Z 690.627,A -85,B 0,C 180,E1 22150.953,E2 22150.953} C_VEL
LIN {X 0,Y 461.184,Z 705.684,A -85,B 0,C 180,E1 22148.73,E2 22148.73} C_VEL
LIN {X 0,Y 459.397,Z 720.651,A -85,B 0,C 180,E1 22146.124,E2 22146.124} C_VEL
LIN {X 0,Y 458.147,Z 732.886,A -85,B 0,C 180,E1 22143.63,E2 22143.63} C_VEL
LIN {X 0,Y 457.165,Z 744.102,A -85,B 0,C 180,E1 22140.879,E2 22140.879} C_VEL
LIN {X 0,Y 456.555,Z 752.934,A -85,B 0,C 180,E1 22138.245,E2 22138.245} C_VEL
LIN {X 0,Y 456.179,Z 760.312,A -85,B 0,C 180,E1 22135.476,E2 22135.476} C_VEL
LIN {X 0,Y 455.998,Z 765.725,A -85,B 0,C 180,E1 22132.822,E2 22132.822} C_VEL
LIN {X 0,Y 455.919,Z 769.527,A -85,B 0,C 180,E1 22130.153,E2 22130.153} C_VEL
LIN {X 0,Y 455.907,Z 771.831,A -85,B 0,C 180,E1 22127.408,E2 22127.408} C_VEL
LIN {X 0,Y 455.907,Z 772.477,A -85,B 0,C 180,E1 22124.744,E2 22124.744} C_VEL
LIN {X 0,Y 455.91,Z 771.515,A -85,B 0,C 180,E1 22121.99,E2 22121.99} C_VEL
LIN {X 0,Y 455.934,Z 769.041,A -85,B 0,C 180,E1 22119.327,E2 22119.327} C_VEL
LIN {X 0,Y 456.013,Z 764.881,A -85,B 0,C 180,E1 22116.62,E2 22116.62} C_VEL
LIN {X 0,Y 456.228,Z 758.954,A -85,B 0,C 180,E1 22113.866,E2 22113.866} C_VEL
LIN {X 0,Y 456.638,Z 751.517,A -85,B 0,C 180,E1 22111.205,E2 22111.205} C_VEL
LIN {X 0,Y 457.324,Z 742.107,A -85,B 0,C 180,E1 22108.501,E2 22108.501} C_VEL
LIN {X 0,Y 458.311,Z 731.141,A -85,B 0,C 180,E1 22105.9,E2 22105.9} C_VEL
LIN {X 0,Y 459.717,Z 717.872,A -85,B 0,C 180,E1 22103.269,E2 22103.269} C_VEL
LIN {X 0,Y 461.511,Z 702.925,A -85,B 0,C 180,E1 22100.76,E2 22100.76} C_VEL
LIN {X 0,Y 463.369,Z 688.307,A -85,B 0,C 180,E1 22098.671,E2 22098.671} C_VEL
LIN {X 0,Y 465.564,Z 671.141,A -85,B 0,C 180,E1 22096.592,E2 22096.592} C_VEL
LIN {X 0,Y 467.765,Z 653.59,A -85,B 0,C 180,E1 22094.797,E2 22094.797} C_VEL
LIN {X 0,Y 470.01,Z 634.342,A -85,B 0,C 180,E1 22093.145,E2 22093.145} C_VEL
LIN {X 0,Y 472.181,Z 614.268,A -85,B 0,C 180,E1 22091.713,E2 22091.713} C_VEL
LIN {X 0,Y 474.089,Z 594.466,A -85,B 0,C 180,E1 22090.549,E2 22090.549} C_VEL
LIN {X 0,Y 475.805,Z 572.899,A -85,B 0,C 180,E1 22089.541,E2 22089.541} C_VEL
LIN {X 0,Y 477.17,Z 551.653,A -85,B 0,C 180,E1 22088.785,E2 22088.785} C_VEL
LIN {X 0,Y 478.209,Z 529.813,A -85,B 0,C 180,E1 22088.223,E2 22088.223} C_VEL
LIN {X 0,Y 480.507,Z 433.338,A -85,B 0,C 180,E1 22086.573,E2 22086.573} C_VEL
LIN {X 0,Y 479.891,Z 425.78,A -85,B 0,C 180,E1 22086.372,E2 22086.372} C_VEL
LIN {X 0,Y 475.368,Z 406.108,A -85,B 0,C 180,E1 22085.572,E2 22085.572} C_VEL
LIN {X 0,Y 474.967,Z 399.609,A -85,B 0,C 180,E1 22085.404,E2 22085.404} C_VEL
LIN {X 0,Y 477.698,Z 300.722,A -85,B 0,C 180,E1 22083.635,E2 22083.635} C_VEL
LIN {X 0,Y 464.733,Z 280.594,A -85,B 0,C 180,E1 22081.775,E2 22081.775} C_VEL
LIN {X 0,Y 455.109,Z 266.652,A -85,B 0,C 180,E1 22080.316,E2 22080.316} C_VEL
LIN {X 0,Y 452.547,Z 262.63,A -85,B 0,C 180,E1 22079.902,E2 22079.902} C_VEL
LIN {X 0,Y 449.831,Z 259.196,A -85,B 0,C 180,E1 22079.477,E2 22079.477} C_VEL
LIN {X 0,Y 449.142,Z 256.791,A -85,B 0,C 180,E1 22079.325,E2 22079.325} C_VEL
LIN {X 0,Y 449.121,Z 256.791,A -85,B 0,C 180,E1 22075.589,E2 22075.589} C_VEL
LIN {X 0,Y 449.098,Z 256.793,A -85,B 0,C 180,E1 22071.965,E2 22071.965} C_VEL
LIN {X 0,Y 449.098,Z 256.793,A -85,B 0,C 180,E1 22068.162,E2 22068.162} C_VEL
LIN {X 0,Y 449.108,Z 256.789,A -85,B 0,C 180,E1 22064.44,E2 22064.44} C_VEL
LIN {X 0,Y 449.131,Z 256.787,A -85,B 0,C 180,E1 22060.779,E2 22060.779} C_VEL
LIN {X 0,Y 449.14,Z 256.787,A -85,B 0,C 180,E1 22057.034,E2 22057.034} C_VEL
LIN {X 0,Y 449.108,Z 256.789,A -85,B 0,C 180,E1 22053.32,E2 22053.32} C_VEL
LIN {X 0,Y 449.089,Z 256.786,A -85,B 0,C 180,E1 22049.746,E2 22049.746} C_VEL
LIN {X 0,Y 449.093,Z 256.783,A -85,B 0,C 180,E1 22046.044,E2 22046.044} C_VEL
LIN {X 0,Y 449.126,Z 256.783,A -85,B 0,C 180,E1 22042.454,E2 22042.454} C_VEL
LIN {X 0,Y 449.131,Z 256.784,A -85,B 0,C 180,E1 22038.704,E2 22038.704} C_VEL
LIN {X 0,Y 449.105,Z 256.788,A -85,B 0,C 180,E1 22035.035,E2 22035.035} C_VEL
LIN {X 0,Y 449.084,Z 256.791,A -85,B 0,C 180,E1 22031.437,E2 22031.437} C_VEL
LIN {X 0,Y 449.082,Z 256.792,A -85,B 0,C 180,E1 22027.623,E2 22027.623} C_VEL
LIN {X 0,Y 449.102,Z 256.794,A -85,B 0,C 180,E1 22023.988,E2 22023.988} C_VEL
LIN {X 0,Y 449.139,Z 256.787,A -85,B 0,C 180,E1 22020.384,E2 22020.384} C_VEL
LIN {X 0,Y 449.113,Z 256.786,A -85,B 0,C 180,E1 22016.596,E2 22016.596} C_VEL
LIN {X 0,Y 449.079,Z 256.788,A -85,B 0,C 180,E1 22013.05,E2 22013.05} C_VEL
LIN {X 0,Y 449.076,Z 256.792,A -85,B 0,C 180,E1 22009.392,E2 22009.392} C_VEL
LIN {X 0,Y 449.102,Z 256.795,A -85,B 0,C 180,E1 22005.794,E2 22005.794} C_VEL
LIN {X 0,Y 449.126,Z 256.794,A -85,B 0,C 180,E1 22002.071,E2 22002.071} C_VEL
LIN {X 0,Y 449.102,Z 256.788,A -85,B 0,C 180,E1 21998.397,E2 21998.397} C_VEL
LIN {X 0,Y 449.073,Z 256.788,A -85,B 0,C 180,E1 21994.746,E2 21994.746} C_VEL
LIN {X 0,Y 449.067,Z 256.791,A -85,B 0,C 180,E1 21990.999,E2 21990.999} C_VEL
LIN {X 0,Y 449.086,Z 256.793,A -85,B 0,C 180,E1 21987.441,E2 21987.441} C_VEL
LIN {X 0,Y 449.117,Z 256.793,A -85,B 0,C 180,E1 21983.761,E2 21983.761} C_VEL
LIN {X 0,Y 449.088,Z 256.792,A -85,B 0,C 180,E1 21980.185,E2 21980.185} C_VEL
LIN {X 0,Y 449.063,Z 256.794,A -85,B 0,C 180,E1 21976.556,E2 21976.556} C_VEL
LIN {X 0,Y 449.06,Z 256.796,A -85,B 0,C 180,E1 21972.787,E2 21972.787} C_VEL
LIN {X 0,Y 449.073,Z 256.796,A -85,B 0,C 180,E1 21969.094,E2 21969.094} C_VEL
LIN {X 0,Y 449.107,Z 256.796,A -85,B 0,C 180,E1 21965.492,E2 21965.492} C_VEL
LIN {X 0,Y 449.094,Z 256.796,A -85,B 0,C 180,E1 21961.784,E2 21961.784} C_VEL
LIN {X 0,Y 449.062,Z 256.796,A -85,B 0,C 180,E1 21958.212,E2 21958.212} C_VEL
LIN {X 0,Y 449.059,Z 256.791,A -85,B 0,C 180,E1 21954.504,E2 21954.504} C_VEL
LIN {X 0,Y 449.081,Z 256.795,A -85,B 0,C 180,E1 21950.903,E2 21950.903} C_VEL
LIN {X 0,Y 449.118,Z 256.792,A -85,B 0,C 180,E1 21947.266,E2 21947.266} C_VEL
LIN {X 0,Y 449.092,Z 256.792,A -85,B 0,C 180,E1 21943.647,E2 21943.647} C_VEL
LIN {X 0,Y 449.068,Z 256.794,A -85,B 0,C 180,E1 21940.082,E2 21940.082} C_VEL
LIN {X 0,Y 449.071,Z 256.792,A -85,B 0,C 180,E1 21936.372,E2 21936.372} C_VEL
LIN {X 0,Y 449.107,Z 256.789,A -85,B 0,C 180,E1 21932.844,E2 21932.844} C_VEL
LIN {X 0,Y 449.122,Z 256.792,A -85,B 0,C 180,E1 21929.199,E2 21929.199} C_VEL
LIN {X 0,Y 449.087,Z 256.796,A -85,B 0,C 180,E1 21925.561,E2 21925.561} C_VEL
LIN {X 0,Y 449.074,Z 256.794,A -85,B 0,C 180,E1 21921.921,E2 21921.921} C_VEL
LIN {X 0,Y 449.1,Z 256.917,A -85,B 0,C 180,E1 21920.309,E2 21920.309} C_VEL
LIN {X 0,Y 450.454,Z 260.385,A -85,B 0,C 180,E1 21919.764,E2 21919.764} C_VEL
LIN {X 0,Y 451.577,Z 262.604,A -85,B 0,C 180,E1 21919.385,E2 21919.385} C_VEL
LIN {X 0,Y 459.1,Z 278.319,A -85,B 0,C 180,E1 21916.849,E2 21916.849} C_VEL
LIN {X 0,Y 466.845,Z 295.72,A -85,B 0,C 180,E1 21914.281,E2 21914.281} C_VEL
LIN {X 0,Y 468.061,Z 298.272,A -85,B 0,C 180,E1 21913.976,E2 21913.976} C_VEL
LIN {X 0,Y 475.024,Z 310.496,A -85,B 0,C 180,E1 21912.926,E2 21912.926} C_VEL
LIN {X 0,Y 478.561,Z 334.22,A -85,B 0,C 180,E1 21912.03,E2 21912.03} C_VEL
LIN {X 0,Y 473.196,Z 529.214,A -85,B 0,C 180,E1 21908.606,E2 21908.606} C_VEL
LIN {X 0,Y 471.142,Z 606.917,A -85,B 0,C 180,E1 21907.237,E2 21907.237} C_VEL
LIN {X 0,Y 469.856,Z 628.943,A -85,B 0,C 180,E1 21906.643,E2 21906.643} C_VEL
LIN {X 0,Y 468.197,Z 651.251,A -85,B 0,C 180,E1 21905.811,E2 21905.811} C_VEL
LIN {X 0,Y 466.273,Z 672.735,A -85,B 0,C 180,E1 21904.776,E2 21904.776} C_VEL
LIN {X 0,Y 464.209,Z 693.454,A -85,B 0,C 180,E1 21903.533,E2 21903.533} C_VEL
LIN {X 0,Y 462.011,Z 712.949,A -85,B 0,C 180,E1 21902.111,E2 21902.111} C_VEL
LIN {X 0,Y 459.668,Z 732.934,A -85,B 0,C 180,E1 21900.378,E2 21900.378} C_VEL
LIN {X 0,Y 457.538,Z 750.49,A -85,B 0,C 180,E1 21898.591,E2 21898.591} C_VEL
LIN {X 0,Y 455.499,Z 767.149,A -85,B 0,C 180,E1 21896.601,E2 21896.601} C_VEL
LIN {X 0,Y 453.651,Z 782.558,A -85,B 0,C 180,E1 21894.458,E2 21894.458} C_VEL
LIN {X 0,Y 452.077,Z 796.47,A -85,B 0,C 180,E1 21892.221,E2 21892.221} C_VEL
LIN {X 0,Y 450.81,Z 808.412,A -85,B 0,C 180,E1 21889.97,E2 21889.97} C_VEL
LIN {X 0,Y 449.706,Z 819.296,A -85,B 0,C 180,E1 21887.465,E2 21887.465} C_VEL
LIN {X 0,Y 448.896,Z 828.887,A -85,B 0,C 180,E1 21884.831,E2 21884.831} C_VEL
LIN {X 0,Y 448.385,Z 836.531,A -85,B 0,C 180,E1 21882.229,E2 21882.229} C_VEL
LIN {X 0,Y 448.09,Z 843.148,A -85,B 0,C 180,E1 21879.373,E2 21879.373} C_VEL
LIN {X 0,Y 447.954,Z 847.823,A -85,B 0,C 180,E1 21876.664,E2 21876.664} C_VEL
LIN {X 0,Y 447.911,Z 850.787,A -85,B 0,C 180,E1 21873.967,E2 21873.967} C_VEL
LIN {X 0,Y 447.91,Z 852.303,A -85,B 0,C 180,E1 21871.15,E2 21871.15} C_VEL
LIN {X 0,Y 447.903,Z 852.257,A -85,B 0,C 180,E1 21868.592,E2 21868.592} C_VEL
LIN {X 0,Y 447.914,Z 850.667,A -85,B 0,C 180,E1 21865.903,E2 21865.903} C_VEL
LIN {X 0,Y 447.962,Z 847.63,A -85,B 0,C 180,E1 21863.205,E2 21863.205} C_VEL
LIN {X 0,Y 448.09,Z 843.142,A -85,B 0,C 180,E1 21860.624,E2 21860.624} C_VEL
LIN {X 0,Y 448.385,Z 836.523,A -85,B 0,C 180,E1 21857.769,E2 21857.769} C_VEL
LIN {X 0,Y 448.9,Z 828.848,A -85,B 0,C 180,E1 21855.157,E2 21855.157} C_VEL
LIN {X 0,Y 449.712,Z 819.231,A -85,B 0,C 180,E1 21852.519,E2 21852.519} C_VEL
LIN {X 0,Y 450.812,Z 808.4,A -85,B 0,C 180,E1 21850.027,E2 21850.027} C_VEL
LIN {X 0,Y 451.939,Z 797.368,A -85,B 0,C 180,E1 21847.971,E2 21847.971} C_VEL
LIN {X 0,Y 453.519,Z 782.731,A -85,B 0,C 180,E1 21845.651,E2 21845.651} C_VEL
LIN {X 0,Y 455.278,Z 767.046,A -85,B 0,C 180,E1 21843.523,E2 21843.523} C_VEL
LIN {X 0,Y 457.206,Z 749.79,A -85,B 0,C 180,E1 21841.526,E2 21841.526} C_VEL
LIN {X 0,Y 459.219,Z 731.539,A -85,B 0,C 180,E1 21839.731,E2 21839.731} C_VEL
LIN {X 0,Y 461.308,Z 711.67,A -85,B 0,C 180,E1 21838.071,E2 21838.071} C_VEL
LIN {X 0,Y 463.27,Z 691.944,A -85,B 0,C 180,E1 21836.682,E2 21836.682} C_VEL
LIN {X 0,Y 465.071,Z 671.384,A -85,B 0,C 180,E1 21835.493,E2 21835.493} C_VEL
LIN {X 0,Y 466.84,Z 649.122,A -85,B 0,C 180,E1 21834.451,E2 21834.451} C_VEL
LIN {X 0,Y 468.338,Z 627.009,A -85,B 0,C 180,E1 21833.645,E2 21833.645} C_VEL
LIN {X 0,Y 469.567,Z 604.005,A -85,B 0,C 180,E1 21833.038,E2 21833.038} C_VEL
LIN {X 0,Y 470.806,Z 550.607,A -85,B 0,C 180,E1 21832.104,E2 21832.104} C_VEL
LIN {X 0,Y 473.943,Z 433.999,A -85,B 0,C 180,E1 21830.021,E2 21830.021} C_VEL
LIN {X 0,Y 477.836,Z 332.601,A -85,B 0,C 180,E1 21828.03,E2 21828.03} C_VEL
LIN {X 0,Y 474.793,Z 308.647,A -85,B 0,C 180,E1 21827.016,E2 21827.016} C_VEL
LIN {X 0,Y 466.884,Z 292.331,A -85,B 0,C 180,E1 21825.404,E2 21825.404} C_VEL
LIN {X 0,Y 462.572,Z 284.141,A -85,B 0,C 180,E1 21824.39,E2 21824.39} C_VEL
LIN {X 0,Y 459.922,Z 278.87,A -85,B 0,C 180,E1 21823.619,E2 21823.619} C_VEL
LIN {X 0,Y 456.393,Z 271.008,A -85,B 0,C 180,E1 21821.928,E2 21821.928} C_VEL
LIN {X 0,Y 454.52,Z 267.017,A -85,B 0,C 180,E1 21820.879,E2 21820.879} C_VEL
LIN {X 0,Y 452.279,Z 263.147,A -85,B 0,C 180,E1 21819.507,E2 21819.507} C_VEL
LIN {X 0,Y 451.8,Z 261.82,A -85,B 0,C 180,E1 21819.032,E2 21819.032} C_VEL
LIN {X 0,Y 449.777,Z 259.126,A -85,B 0,C 180,E1 21817.205,E2 21817.205} C_VEL
LIN {X 0,Y 449.247,Z 257.623,A -85,B 0,C 180,E1 21815.358,E2 21815.358} C_VEL
LIN {X 0,Y 449.283,Z 257.874,A -85,B 0,C 180,E1 21814.31,E2 21814.31} C_VEL
LIN {X 0,Y 451.076,Z 261.122,A -85,B 0,C 180,E1 21813.155,E2 21813.155} C_VEL
LIN {X 0,Y 454.203,Z 263.484,A -85,B 0,C 180,E1 21811.937,E2 21811.937} C_VEL
LIN {X 0,Y 456.224,Z 267.213,A -85,B 0,C 180,E1 21811.185,E2 21811.185} C_VEL
LIN {X 0,Y 458.582,Z 269.659,A -85,B 0,C 180,E1 21810.513,E2 21810.513} C_VEL
LIN {X 0,Y 461.395,Z 273.757,A -85,B 0,C 180,E1 21809.753,E2 21809.753} C_VEL
LIN {X 0,Y 463.019,Z 276.193,A -85,B 0,C 180,E1 21809.354,E2 21809.354} C_VEL
LIN {X 0,Y 466.782,Z 281.706,A -85,B 0,C 180,E1 21808.505,E2 21808.505} C_VEL
LIN {X 0,Y 473.067,Z 291.734,A -85,B 0,C 180,E1 21807.259,E2 21807.259} C_VEL
LIN {X 0,Y 478.306,Z 301.419,A -85,B 0,C 180,E1 21806.313,E2 21806.313} C_VEL
LIN {X 0,Y 474.116,Z 401.345,A -85,B 0,C 180,E1 21804.349,E2 21804.349} C_VEL
LIN {X 0,Y 470.91,Z 515.798,A -85,B 0,C 180,E1 21802.289,E2 21802.289} C_VEL
LIN {X 0,Y 470.044,Z 542.863,A -85,B 0,C 180,E1 21801.749,E2 21801.749} C_VEL
LIN {X 0,Y 468.972,Z 564.823,A -85,B 0,C 180,E1 21801.084,E2 21801.084} C_VEL
LIN {X 0,Y 467.587,Z 585.435,A -85,B 0,C 180,E1 21800.247,E2 21800.247} C_VEL
LIN {X 0,Y 465.918,Z 605.126,A -85,B 0,C 180,E1 21799.223,E2 21799.223} C_VEL
LIN {X 0,Y 463.955,Z 625.057,A -85,B 0,C 180,E1 21797.951,E2 21797.951} C_VEL
LIN {X 0,Y 461.857,Z 644.126,A -85,B 0,C 180,E1 21796.476,E2 21796.476} C_VEL
LIN {X 0,Y 459.639,Z 662.01,A -85,B 0,C 180,E1 21794.81,E2 21794.81} C_VEL
LIN {X 0,Y 457.489,Z 678.349,A -85,B 0,C 180,E1 21793.011,E2 21793.011} C_VEL
LIN {X 0,Y 455.409,Z 693.817,A -85,B 0,C 180,E1 21791.013,E2 21791.013} C_VEL
LIN {X 0,Y 453.408,Z 708.605,A -85,B 0,C 180,E1 21788.754,E2 21788.754} C_VEL
LIN {X 0,Y 451.603,Z 722.417,A -85,B 0,C 180,E1 21786.23,E2 21786.23} C_VEL
LIN {X 0,Y 450.232,Z 734.047,A -85,B 0,C 180,E1 21783.694,E2 21783.694} C_VEL
LIN {X 0,Y 449.208,Z 745.101,A -85,B 0,C 180,E1 21780.894,E2 21780.894} C_VEL
LIN {X 0,Y 448.544,Z 754.076,A -85,B 0,C 180,E1 21778.086,E2 21778.086} C_VEL
LIN {X 0,Y 448.163,Z 761.242,A -85,B 0,C 180,E1 21775.267,E2 21775.267} C_VEL
LIN {X 0,Y 447.982,Z 766.566,A -85,B 0,C 180,E1 21772.435,E2 21772.435} C_VEL
LIN {X 0,Y 447.916,Z 770.108,A -85,B 0,C 180,E1 21769.715,E2 21769.715} C_VEL
LIN {X 0,Y 447.905,Z 772.051,A -85,B 0,C 180,E1 21766.972,E2 21766.972} C_VEL
LIN {X 0,Y 447.912,Z 772.408,A -85,B 0,C 180,E1 21764.178,E2 21764.178} C_VEL
LIN {X 0,Y 447.915,Z 771.26,A -85,B 0,C 180,E1 21761.522,E2 21761.522} C_VEL
LIN {X 0,Y 447.94,Z 768.497,A -85,B 0,C 180,E1 21758.804,E2 21758.804} C_VEL
LIN {X 0,Y 448.065,Z 763.788,A -85,B 0,C 180,E1 21755.88,E2 21755.88} C_VEL
LIN {X 0,Y 448.341,Z 757.5,A -85,B 0,C 180,E1 21753.085,E2 21753.085} C_VEL
LIN {X 0,Y 448.879,Z 749.193,A -85,B 0,C 180,E1 21750.219,E2 21750.219} C_VEL
LIN {X 0,Y 449.667,Z 739.77,A -85,B 0,C 180,E1 21747.6,E2 21747.6} C_VEL
LIN {X 0,Y 451.024,Z 727.037,A -85,B 0,C 180,E1 21744.651,E2 21744.651} C_VEL
LIN {X 0,Y 452.686,Z 713.584,A -85,B 0,C 180,E1 21742.048,E2 21742.048} C_VEL
LIN {X 0,Y 454.583,Z 699.175,A -85,B 0,C 180,E1 21739.714,E2 21739.714} C_VEL
LIN {X 0,Y 456.739,Z 683.348,A -85,B 0,C 180,E1 21737.54,E2 21737.54} C_VEL
LIN {X 0,Y 458.977,Z 666.69,A -85,B 0,C 180,E1 21735.606,E2 21735.606} C_VEL
LIN {X 0,Y 461.336,Z 648.429,A -85,B 0,C 180,E1 21733.808,E2 21733.808} C_VEL
LIN {X 0,Y 463.584,Z 630.19,A -85,B 0,C 180,E1 21732.291,E2 21732.291} C_VEL
LIN {X 0,Y 465.64,Z 611.511,A -85,B 0,C 180,E1 21730.999,E2 21730.999} C_VEL
LIN {X 0,Y 467.642,Z 590.822,A -85,B 0,C 180,E1 21729.82,E2 21729.82} C_VEL
LIN {X 0,Y 469.392,Z 569.897,A -85,B 0,C 180,E1 21728.87,E2 21728.87} C_VEL
LIN {X 0,Y 470.697,Z 549.447,A -85,B 0,C 180,E1 21728.163,E2 21728.163} C_VEL
LIN {X 0,Y 471.736,Z 526.892,A -85,B 0,C 180,E1 21727.61,E2 21727.61} C_VEL
LIN {X 0,Y 474.967,Z 399.609,A -85,B 0,C 180,E1 21725.404,E2 21725.404} C_VEL
LIN {X 0,Y 474.43,Z 392.058,A -85,B 0,C 180,E1 21725.197,E2 21725.197} C_VEL
LIN {X 0,Y 470.128,Z 372.411,A -85,B 0,C 180,E1 21724.363,E2 21724.363} C_VEL
LIN {X 0,Y 469.73,Z 365.917,A -85,B 0,C 180,E1 21724.189,E2 21724.189} C_VEL
LIN {X 0,Y 471.587,Z 304.106,A -85,B 0,C 180,E1 21723.058,E2 21723.058} C_VEL
LIN {X 0,Y 457.57,Z 282.462,A -85,B 0,C 180,E1 21720.99,E2 21720.99} C_VEL
LIN {X 0,Y 447.196,Z 267.629,A -85,B 0,C 180,E1 21719.355,E2 21719.355} C_VEL
LIN {X 0,Y 444.653,Z 263.579,A -85,B 0,C 180,E1 21718.931,E2 21718.931} C_VEL
LIN {X 0,Y 441.933,Z 260.334,A -85,B 0,C 180,E1 21718.497,E2 21718.497} C_VEL
LIN {X 0,Y 441.163,Z 257.784,A -85,B 0,C 180,E1 21718.309,E2 21718.309} C_VEL
LIN {X 0,Y 441.178,Z 257.779,A -85,B 0,C 180,E1 21714.647,E2 21714.647} C_VEL
LIN {X 0,Y 441.2,Z 257.775,A -85,B 0,C 180,E1 21710.982,E2 21710.982} C_VEL
LIN {X 0,Y 441.191,Z 257.779,A -85,B 0,C 180,E1 21707.271,E2 21707.271} C_VEL
LIN {X 0,Y 441.164,Z 257.775,A -85,B 0,C 180,E1 21703.634,E2 21703.634} C_VEL
LIN {X 0,Y 441.156,Z 257.781,A -85,B 0,C 180,E1 21699.92,E2 21699.92} C_VEL
LIN {X 0,Y 441.157,Z 257.777,A -85,B 0,C 180,E1 21696.116,E2 21696.116} C_VEL
LIN {X 0,Y 441.177,Z 257.773,A -85,B 0,C 180,E1 21692.469,E2 21692.469} C_VEL
LIN {X 0,Y 441.198,Z 257.769,A -85,B 0,C 180,E1 21688.833,E2 21688.833} C_VEL
LIN {X 0,Y 441.177,Z 257.768,A -85,B 0,C 180,E1 21685.061,E2 21685.061} C_VEL
LIN {X 0,Y 441.151,Z 257.774,A -85,B 0,C 180,E1 21681.53,E2 21681.53} C_VEL
LIN {X 0,Y 441.148,Z 257.777,A -85,B 0,C 180,E1 21677.7,E2 21677.7} C_VEL
LIN {X 0,Y 441.163,Z 257.776,A -85,B 0,C 180,E1 21674.085,E2 21674.085} C_VEL
LIN {X 0,Y 441.189,Z 257.773,A -85,B 0,C 180,E1 21670.404,E2 21670.404} C_VEL
LIN {X 0,Y 441.175,Z 257.779,A -85,B 0,C 180,E1 21666.777,E2 21666.777} C_VEL
LIN {X 0,Y 441.145,Z 257.781,A -85,B 0,C 180,E1 21663.192,E2 21663.192} C_VEL
LIN {X 0,Y 441.142,Z 257.783,A -85,B 0,C 180,E1 21659.455,E2 21659.455} C_VEL
LIN {X 0,Y 441.156,Z 257.785,A -85,B 0,C 180,E1 21655.802,E2 21655.802} C_VEL
LIN {X 0,Y 441.181,Z 257.778,A -85,B 0,C 180,E1 21652.058,E2 21652.058} C_VEL
LIN {X 0,Y 441.18,Z 257.776,A -85,B 0,C 180,E1 21648.394,E2 21648.394} C_VEL
LIN {X 0,Y 441.144,Z 257.783,A -85,B 0,C 180,E1 21644.815,E2 21644.815} C_VEL
LIN {X 0,Y 441.132,Z 257.785,A -85,B 0,C 180,E1 21641.091,E2 21641.091} C_VEL
LIN {X 0,Y 441.141,Z 257.785,A -85,B 0,C 180,E1 21637.401,E2 21637.401} C_VEL
LIN {X 0,Y 441.165,Z 257.781,A -85,B 0,C 180,E1 21633.723,E2 21633.723} C_VEL
LIN {X 0,Y 441.19,Z 257.773,A -85,B 0,C 180,E1 21629.903,E2 21629.903} C_VEL
LIN {X 0,Y 441.161,Z 257.778,A -85,B 0,C 180,E1 21626.173,E2 21626.173} C_VEL
LIN {X 0,Y 441.131,Z 257.783,A -85,B 0,C 180,E1 21622.52,E2 21622.52} C_VEL
LIN {X 0,Y 441.123,Z 257.783,A -85,B 0,C 180,E1 21618.773,E2 21618.773} C_VEL
LIN {X 0,Y 441.132,Z 257.782,A -85,B 0,C 180,E1 21615.088,E2 21615.088} C_VEL
LIN {X 0,Y 441.162,Z 257.78,A -85,B 0,C 180,E1 21611.502,E2 21611.502} C_VEL
LIN {X 0,Y 441.177,Z 257.779,A -85,B 0,C 180,E1 21607.682,E2 21607.682} C_VEL
LIN {X 0,Y 441.147,Z 257.782,A -85,B 0,C 180,E1 21603.897,E2 21603.897} C_VEL
LIN {X 0,Y 441.122,Z 257.78,A -85,B 0,C 180,E1 21600.258,E2 21600.258} C_VEL
LIN {X 0,Y 441.119,Z 257.785,A -85,B 0,C 180,E1 21596.49,E2 21596.49} C_VEL
LIN {X 0,Y 441.133,Z 257.784,A -85,B 0,C 180,E1 21592.837,E2 21592.837} C_VEL
LIN {X 0,Y 441.173,Z 257.779,A -85,B 0,C 180,E1 21589.288,E2 21589.288} C_VEL
LIN {X 0,Y 441.162,Z 257.779,A -85,B 0,C 180,E1 21585.562,E2 21585.562} C_VEL
LIN {X 0,Y 441.134,Z 257.784,A -85,B 0,C 180,E1 21581.908,E2 21581.908} C_VEL
LIN {X 0,Y 441.128,Z 257.782,A -85,B 0,C 180,E1 21578.177,E2 21578.177} C_VEL
LIN {X 0,Y 441.135,Z 257.78,A -85,B 0,C 180,E1 21574.43,E2 21574.43} C_VEL
LIN {X 0,Y 441.171,Z 257.778,A -85,B 0,C 180,E1 21570.837,E2 21570.837} C_VEL
LIN {X 0,Y 441.177,Z 257.78,A -85,B 0,C 180,E1 21567.202,E2 21567.202} C_VEL
LIN {X 0,Y 441.146,Z 257.783,A -85,B 0,C 180,E1 21563.569,E2 21563.569} C_VEL
LIN {X 0,Y 441.192,Z 257.968,A -85,B 0,C 180,E1 21561.281,E2 21561.281} C_VEL
LIN {X 0,Y 442.464,Z 261.233,A -85,B 0,C 180,E1 21560.747,E2 21560.747} C_VEL
LIN {X 0,Y 443.557,Z 263.426,A -85,B 0,C 180,E1 21560.361,E2 21560.361} C_VEL
LIN {X 0,Y 449.852,Z 276.384,A -85,B 0,C 180,E1 21558.179,E2 21558.179} C_VEL
LIN {X 0,Y 457.631,Z 293.267,A -85,B 0,C 180,E1 21555.552,E2 21555.552} C_VEL
LIN {X 0,Y 459.512,Z 297.331,A -85,B 0,C 180,E1 21554.994,E2 21554.994} C_VEL
LIN {X 0,Y 469.387,Z 314.265,A -85,B 0,C 180,E1 21553.467,E2 21553.467} C_VEL
LIN {X 0,Y 472.52,Z 335.79,A -85,B 0,C 180,E1 21552.645,E2 21552.645} C_VEL
LIN {X 0,Y 466.819,Z 526.083,A -85,B 0,C 180,E1 21549.239,E2 21549.239} C_VEL
LIN {X 0,Y 464.544,Z 606.429,A -85,B 0,C 180,E1 21547.801,E2 21547.801} C_VEL
LIN {X 0,Y 463.164,Z 628.615,A -85,B 0,C 180,E1 21547.194,E2 21547.194} C_VEL
LIN {X 0,Y 461.456,Z 650.283,A -85,B 0,C 180,E1 21546.377,E2 21546.377} C_VEL
LIN {X 0,Y 459.48,Z 671.23,A -85,B 0,C 180,E1 21545.366,E2 21545.366} C_VEL
LIN {X 0,Y 457.309,Z 691.777,A -85,B 0,C 180,E1 21544.126,E2 21544.126} C_VEL
LIN {X 0,Y 454.949,Z 711.613,A -85,B 0,C 180,E1 21542.675,E2 21542.675} C_VEL
LIN {X 0,Y 452.447,Z 731.757,A -85,B 0,C 180,E1 21540.915,E2 21540.915} C_VEL
LIN {X 0,Y 450.181,Z 749.402,A -85,B 0,C 180,E1 21539.102,E2 21539.102} C_VEL
LIN {X 0,Y 447.985,Z 766.276,A -85,B 0,C 180,E1 21537.059,E2 21537.059} C_VEL
LIN {X 0,Y 446.042,Z 781.453,A -85,B 0,C 180,E1 21534.923,E2 21534.923} C_VEL
LIN {X 0,Y 444.345,Z 795.552,A -85,B 0,C 180,E1 21532.628,E2 21532.628} C_VEL
LIN {X 0,Y 442.927,Z 808.212,A -85,B 0,C 180,E1 21530.203,E2 21530.203} C_VEL
LIN {X 0,Y 441.798,Z 819.518,A -85,B 0,C 180,E1 21527.652,E2 21527.652} C_VEL
LIN {X 0,Y 441.106,Z 827.513,A -85,B 0,C 180,E1 21525.512,E2 21525.512} C_VEL
LIN {X 0,Y 440.502,Z 835.471,A -85,B 0,C 180,E1 21522.851,E2 21522.851} C_VEL
LIN {X 0,Y 440.158,Z 841.875,A -85,B 0,C 180,E1 21520.204,E2 21520.204} C_VEL
LIN {X 0,Y 439.985,Z 846.814,A -85,B 0,C 180,E1 21517.441,E2 21517.441} C_VEL
LIN {X 0,Y 439.922,Z 850.332,A -85,B 0,C 180,E1 21514.561,E2 21514.561} C_VEL
LIN {X 0,Y 439.905,Z 852.086,A -85,B 0,C 180,E1 21511.952,E2 21511.952} C_VEL
LIN {X 0,Y 439.904,Z 852.37,A -85,B 0,C 180,E1 21509.217,E2 21509.217} C_VEL
LIN {X 0,Y 439.911,Z 851.234,A -85,B 0,C 180,E1 21506.48,E2 21506.48} C_VEL
LIN {X 0,Y 439.943,Z 848.614,A -85,B 0,C 180,E1 21503.867,E2 21503.867} C_VEL
LIN {X 0,Y 440.047,Z 844.412,A -85,B 0,C 180,E1 21501.111,E2 21501.111} C_VEL
LIN {X 0,Y 440.302,Z 838.853,A -85,B 0,C 180,E1 21498.472,E2 21498.472} C_VEL
LIN {X 0,Y 440.797,Z 831.28,A -85,B 0,C 180,E1 21495.684,E2 21495.684} C_VEL
LIN {X 0,Y 441.481,Z 823.267,A -85,B 0,C 180,E1 21493.283,E2 21493.283} C_VEL
LIN {X 0,Y 442.468,Z 812.402,A -85,B 0,C 180,E1 21490.735,E2 21490.735} C_VEL
LIN {X 0,Y 443.796,Z 799.429,A -85,B 0,C 180,E1 21488.176,E2 21488.176} C_VEL
LIN {X 0,Y 445.336,Z 785.746,A -85,B 0,C 180,E1 21485.881,E2 21485.881} C_VEL
LIN {X 0,Y 447.155,Z 770.05,A -85,B 0,C 180,E1 21483.649,E2 21483.649} C_VEL
LIN {X 0,Y 449.19,Z 752.776,A -85,B 0,C 180,E1 21481.551,E2 21481.551} C_VEL
LIN {X 0,Y 451.313,Z 734.513,A -85,B 0,C 180,E1 21479.66,E2 21479.66} C_VEL
LIN {X 0,Y 453.507,Z 714.984,A -85,B 0,C 180,E1 21477.947,E2 21477.947} C_VEL
LIN {X 0,Y 455.554,Z 695.163,A -85,B 0,C 180,E1 21476.495,E2 21476.495} C_VEL
LIN {X 0,Y 457.664,Z 673.148,A -85,B 0,C 180,E1 21475.158,E2 21475.158} C_VEL
LIN {X 0,Y 459.53,Z 651.665,A -85,B 0,C 180,E1 21474.098,E2 21474.098} C_VEL
LIN {X 0,Y 461.133,Z 629.937,A -85,B 0,C 180,E1 21473.262,E2 21473.262} C_VEL
LIN {X 0,Y 462.506,Z 606.805,A -85,B 0,C 180,E1 21472.607,E2 21472.607} C_VEL
LIN {X 0,Y 463.497,Z 575.717,A -85,B 0,C 180,E1 21472.008,E2 21472.008} C_VEL
LIN {X 0,Y 466.592,Z 463.401,A -85,B 0,C 180,E1 21469.98,E2 21469.98} C_VEL
LIN {X 0,Y 470.756,Z 360.336,A -85,B 0,C 180,E1 21467.939,E2 21467.939} C_VEL
LIN {X 0,Y 471.956,Z 333.736,A -85,B 0,C 180,E1 21467.366,E2 21467.366} C_VEL
LIN {X 0,Y 469.587,Z 312.785,A -85,B 0,C 180,E1 21466.448,E2 21466.448} C_VEL
LIN {X 0,Y 462.539,Z 297.63,A -85,B 0,C 180,E1 21464.894,E2 21464.894} C_VEL
LIN {X 0,Y 457.443,Z 287.454,A -85,B 0,C 180,E1 21463.557,E2 21463.557} C_VEL
LIN {X 0,Y 452.967,Z 279.581,A -85,B 0,C 180,E1 21462.148,E2 21462.148} C_VEL
LIN {X 0,Y 450.82,Z 275.935,A -85,B 0,C 180,E1 21461.329,E2 21461.329} C_VEL
LIN {X 0,Y 449.031,Z 272.499,A -85,B 0,C 180,E1 21460.474,E2 21460.474} C_VEL
LIN {X 0,Y 447.269,Z 269.039,A -85,B 0,C 180,E1 21459.246,E2 21459.246} C_VEL
LIN {X 0,Y 446.774,Z 268.011,A -85,B 0,C 180,E1 21458.803,E2 21458.803} C_VEL
LIN {X 0,Y 445.643,Z 266.441,A -85,B 0,C 180,E1 21457.61,E2 21457.61} C_VEL
LIN {X 0,Y 445.754,Z 265.236,A -85,B 0,C 180,E1 21456.146,E2 21456.146} C_VEL
LIN {X 0,Y 446.96,Z 265.261,A -85,B 0,C 180,E1 21454.782,E2 21454.782} C_VEL
LIN {X 0,Y 447.426,Z 265.962,A -85,B 0,C 180,E1 21454.391,E2 21454.391} C_VEL
LIN {X 0,Y 449.639,Z 269.368,A -85,B 0,C 180,E1 21453.035,E2 21453.035} C_VEL
LIN {X 0,Y 451.695,Z 271.109,A -85,B 0,C 180,E1 21452.205,E2 21452.205} C_VEL
LIN {X 0,Y 454.192,Z 275.127,A -85,B 0,C 180,E1 21451.273,E2 21451.273} C_VEL
LIN {X 0,Y 455.677,Z 276.893,A -85,B 0,C 180,E1 21450.821,E2 21450.821} C_VEL
LIN {X 0,Y 459.382,Z 282.421,A -85,B 0,C 180,E1 21449.784,E2 21449.784} C_VEL
LIN {X 0,Y 464.16,Z 289.701,A -85,B 0,C 180,E1 21448.652,E2 21448.652} C_VEL
LIN {X 0,Y 470.498,Z 300.698,A -85,B 0,C 180,E1 21447.339,E2 21447.339} C_VEL
LIN {X 0,Y 472.585,Z 304.82,A -85,B 0,C 180,E1 21446.944,E2 21446.944} C_VEL
LIN {X 0,Y 467.975,Z 400.746,A -85,B 0,C 180,E1 21444.986,E2 21444.986} C_VEL
LIN {X 0,Y 464.529,Z 506.625,A -85,B 0,C 180,E1 21443.005,E2 21443.005} C_VEL
LIN {X 0,Y 463.45,Z 541.228,A -85,B 0,C 180,E1 21442.338,E2 21442.338} C_VEL
LIN {X 0,Y 462.349,Z 563.556,A -85,B 0,C 180,E1 21441.679,E2 21441.679} C_VEL
LIN {X 0,Y 460.908,Z 584.223,A -85,B 0,C 180,E1 21440.842,E2 21440.842} C_VEL
LIN {X 0,Y 459.145,Z 604.559,A -85,B 0,C 180,E1 21439.794,E2 21439.794} C_VEL
LIN {X 0,Y 457.162,Z 624.115,A -85,B 0,C 180,E1 21438.557,E2 21438.557} C_VEL
LIN {X 0,Y 455.041,Z 642.679,A -85,B 0,C 180,E1 21437.125,E2 21437.125} C_VEL
LIN {X 0,Y 452.757,Z 660.347,A -85,B 0,C 180,E1 21435.5,E2 21435.5} C_VEL
LIN {X 0,Y 450.494,Z 677.165,A -85,B 0,C 180,E1 21433.674,E2 21433.674} C_VEL
LIN {X 0,Y 448.316,Z 692.522,A -85,B 0,C 180,E1 21431.711,E2 21431.711} C_VEL
LIN {X 0,Y 446.259,Z 706.828,A -85,B 0,C 180,E1 21429.545,E2 21429.545} C_VEL
LIN {X 0,Y 444.351,Z 720.517,A -85,B 0,C 180,E1 21427.103,E2 21427.103} C_VEL
LIN {X 0,Y 442.787,Z 732.578,A -85,B 0,C 180,E1 21424.535,E2 21424.535} C_VEL
LIN {X 0,Y 441.616,Z 742.657,A -85,B 0,C 180,E1 21421.948,E2 21421.948} C_VEL
LIN {X 0,Y 440.681,Z 753.018,A -85,B 0,C 180,E1 21418.702,E2 21418.702} C_VEL
LIN {X 0,Y 440.236,Z 760.379,A -85,B 0,C 180,E1 21415.834,E2 21415.834} C_VEL
LIN {X 0,Y 440.02,Z 765.767,A -85,B 0,C 180,E1 21413.085,E2 21413.085} C_VEL
LIN {X 0,Y 439.922,Z 769.691,A -85,B 0,C 180,E1 21410.187,E2 21410.187} C_VEL
LIN {X 0,Y 439.907,Z 771.887,A -85,B 0,C 180,E1 21407.399,E2 21407.399} C_VEL
LIN {X 0,Y 439.907,Z 772.474,A -85,B 0,C 180,E1 21404.715,E2 21404.715} C_VEL
LIN {X 0,Y 439.91,Z 771.5,A -85,B 0,C 180,E1 21401.86,E2 21401.86} C_VEL
LIN {X 0,Y 439.942,Z 768.998,A -85,B 0,C 180,E1 21399.082,E2 21399.082} C_VEL
LIN {X 0,Y 440.034,Z 764.829,A -85,B 0,C 180,E1 21396.288,E2 21396.288} C_VEL
LIN {X 0,Y 440.307,Z 758.885,A -85,B 0,C 180,E1 21393.429,E2 21393.429} C_VEL
LIN {X 0,Y 440.796,Z 751.409,A -85,B 0,C 180,E1 21390.665,E2 21390.665} C_VEL
LIN {X 0,Y 441.697,Z 741.676,A -85,B 0,C 180,E1 21387.711,E2 21387.711} C_VEL
LIN {X 0,Y 442.939,Z 730.798,A -85,B 0,C 180,E1 21385.018,E2 21385.018} C_VEL
LIN {X 0,Y 444.548,Z 718.358,A -85,B 0,C 180,E1 21382.448,E2 21382.448} C_VEL
LIN {X 0,Y 446.521,Z 704.055,A -85,B 0,C 180,E1 21379.98,E2 21379.98} C_VEL
LIN {X 0,Y 448.75,Z 688.482,A -85,B 0,C 180,E1 21377.709,E2 21377.709} C_VEL
LIN {X 0,Y 451.123,Z 671.949,A -85,B 0,C 180,E1 21375.661,E2 21375.661} C_VEL
LIN {X 0,Y 453.617,Z 654.109,A -85,B 0,C 180,E1 21373.799,E2 21373.799} C_VEL
LIN {X 0,Y 456.001,Z 635.606,A -85,B 0,C 180,E1 21372.177,E2 21372.177} C_VEL
LIN {X 0,Y 458.413,Z 615.49,A -85,B 0,C 180,E1 21370.705,E2 21370.705} C_VEL
LIN {X 0,Y 460.425,Z 596.756,A -85,B 0,C 180,E1 21369.568,E2 21369.568} C_VEL
LIN {X 0,Y 462.256,Z 575.934,A -85,B 0,C 180,E1 21368.557,E2 21368.557} C_VEL
LIN {X 0,Y 463.877,Z 553.717,A -85,B 0,C 180,E1 21367.727,E2 21367.727} C_VEL
LIN {X 0,Y 465.044,Z 532.232,A -85,B 0,C 180,E1 21367.146,E2 21367.146} C_VEL
LIN {X 0,Y 469.73,Z 365.917,A -85,B 0,C 180,E1 21364.189,E2 21364.189} C_VEL
LIN {X 0,Y 469.203,Z 358.368,A -85,B 0,C 180,E1 21363.975,E2 21363.975} C_VEL
LIN {X 0,Y 465.115,Z 338.727,A -85,B 0,C 180,E1 21363.115,E2 21363.115} C_VEL
LIN {X 0,Y 464.779,Z 332.237,A -85,B 0,C 180,E1 21362.937,E2 21362.937} C_VEL
LIN {X 0,Y 465.447,Z 307.497,A -85,B 0,C 180,E1 21362.465,E2 21362.465} C_VEL
LIN {X 0,Y 452.605,Z 287.672,A -85,B 0,C 180,E1 21360.52,E2 21360.52} C_VEL
LIN {X 0,Y 442.323,Z 272.979,A -85,B 0,C 180,E1 21358.876,E2 21358.876} C_VEL
LIN {X 0,Y 439.451,Z 268.819,A -85,B 0,C 180,E1 21358.395,E2 21358.395} C_VEL
LIN {X 0,Y 436.82,Z 264.781,A -85,B 0,C 180,E1 21357.937,E2 21357.937} C_VEL
LIN {X 0,Y 433.99,Z 261.254,A -85,B 0,C 180,E1 21357.457,E2 21357.457} C_VEL
LIN {X 0,Y 433.263,Z 258.764,A -85,B 0,C 180,E1 21357.252,E2 21357.252} C_VEL
LIN {X 0,Y 433.255,Z 258.765,A -85,B 0,C 180,E1 21353.388,E2 21353.388} C_VEL
LIN {X 0,Y 433.232,Z 258.77,A -85,B 0,C 180,E1 21349.683,E2 21349.683} C_VEL
LIN {X 0,Y 433.219,Z 258.768,A -85,B 0,C 180,E1 21345.942,E2 21345.942} C_VEL
LIN {X 0,Y 433.219,Z 258.77,A -85,B 0,C 180,E1 21342.125,E2 21342.125} C_VEL
LIN {X 0,Y 433.228,Z 258.765,A -85,B 0,C 180,E1 21338.362,E2 21338.362} C_VEL
LIN {X 0,Y 433.249,Z 258.764,A -85,B 0,C 180,E1 21334.634,E2 21334.634} C_VEL
LIN {X 0,Y 433.262,Z 258.764,A -85,B 0,C 180,E1 21330.795,E2 21330.795} C_VEL
LIN {X 0,Y 433.247,Z 258.765,A -85,B 0,C 180,E1 21326.959,E2 21326.959} C_VEL
LIN {X 0,Y 433.225,Z 258.766,A -85,B 0,C 180,E1 21323.242,E2 21323.242} C_VEL
LIN {X 0,Y 433.212,Z 258.767,A -85,B 0,C 180,E1 21319.469,E2 21319.469} C_VEL
LIN {X 0,Y 433.208,Z 258.768,A -85,B 0,C 180,E1 21315.704,E2 21315.704} C_VEL
LIN {X 0,Y 433.22,Z 258.77,A -85,B 0,C 180,E1 21311.958,E2 21311.958} C_VEL
LIN {X 0,Y 433.254,Z 258.77,A -85,B 0,C 180,E1 21308.333,E2 21308.333} C_VEL
LIN {X 0,Y 433.246,Z 258.766,A -85,B 0,C 180,E1 21304.581,E2 21304.581} C_VEL
LIN {X 0,Y 433.221,Z 258.765,A -85,B 0,C 180,E1 21300.86,E2 21300.86} C_VEL
LIN {X 0,Y 433.203,Z 258.764,A -85,B 0,C 180,E1 21297.149,E2 21297.149} C_VEL
LIN {X 0,Y 433.201,Z 258.766,A -85,B 0,C 180,E1 21293.433,E2 21293.433} C_VEL
LIN {X 0,Y 433.217,Z 258.77,A -85,B 0,C 180,E1 21289.744,E2 21289.744} C_VEL
LIN {X 0,Y 433.243,Z 258.775,A -85,B 0,C 180,E1 21286.054,E2 21286.054} C_VEL
LIN {X 0,Y 433.246,Z 258.77,A -85,B 0,C 180,E1 21282.185,E2 21282.185} C_VEL
LIN {X 0,Y 433.212,Z 258.766,A -85,B 0,C 180,E1 21278.521,E2 21278.521} C_VEL
LIN {X 0,Y 433.192,Z 258.765,A -85,B 0,C 180,E1 21274.916,E2 21274.916} C_VEL
LIN {X 0,Y 433.191,Z 258.769,A -85,B 0,C 180,E1 21271.099,E2 21271.099} C_VEL
LIN {X 0,Y 433.211,Z 258.771,A -85,B 0,C 180,E1 21267.488,E2 21267.488} C_VEL
LIN {X 0,Y 433.24,Z 258.77,A -85,B 0,C 180,E1 21263.818,E2 21263.818} C_VEL
LIN {X 0,Y 433.216,Z 258.77,A -85,B 0,C 180,E1 21260.112,E2 21260.112} C_VEL
LIN {X 0,Y 433.188,Z 258.772,A -85,B 0,C 180,E1 21256.491,E2 21256.491} C_VEL
LIN {X 0,Y 433.184,Z 258.774,A -85,B 0,C 180,E1 21252.8,E2 21252.8} C_VEL
LIN {X 0,Y 433.191,Z 258.774,A -85,B 0,C 180,E1 21249.028,E2 21249.028} C_VEL
LIN {X 0,Y 433.223,Z 258.774,A -85,B 0,C 180,E1 21245.428,E2 21245.428} C_VEL
LIN {X 0,Y 433.231,Z 258.771,A -85,B 0,C 180,E1 21241.585,E2 21241.585} C_VEL
LIN {X 0,Y 433.205,Z 258.773,A -85,B 0,C 180,E1 21237.882,E2 21237.882} C_VEL
LIN {X 0,Y 433.187,Z 258.768,A -85,B 0,C 180,E1 21234.169,E2 21234.169} C_VEL
LIN {X 0,Y 433.184,Z 258.774,A -85,B 0,C 180,E1 21230.432,E2 21230.432} C_VEL
LIN {X 0,Y 433.193,Z 258.77,A -85,B 0,C 180,E1 21226.654,E2 21226.654} C_VEL
LIN {X 0,Y 433.231,Z 258.768,A -85,B 0,C 180,E1 21223.093,E2 21223.093} C_VEL
LIN {X 0,Y 433.24,Z 258.767,A -85,B 0,C 180,E1 21219.321,E2 21219.321} C_VEL
LIN {X 0,Y 433.212,Z 258.77,A -85,B 0,C 180,E1 21215.597,E2 21215.597} C_VEL
LIN {X 0,Y 433.195,Z 258.771,A -85,B 0,C 180,E1 21211.909,E2 21211.909} C_VEL
LIN {X 0,Y 433.195,Z 258.774,A -85,B 0,C 180,E1 21208.091,E2 21208.091} C_VEL
LIN {X 0,Y 433.203,Z 258.775,A -85,B 0,C 180,E1 21204.331,E2 21204.331} C_VEL
LIN {X 0,Y 433.239,Z 259.016,A -85,B 0,C 180,E1 21202.295,E2 21202.295} C_VEL
LIN {X 0,Y 434.49,Z 262.233,A -85,B 0,C 180,E1 21201.754,E2 21201.754} C_VEL
LIN {X 0,Y 435.635,Z 264.245,A -85,B 0,C 180,E1 21201.369,E2 21201.369} C_VEL
LIN {X 0,Y 443.677,Z 280.867,A -85,B 0,C 180,E1 21198.504,E2 21198.504} C_VEL
LIN {X 0,Y 450.817,Z 296.396,A -85,B 0,C 180,E1 21196.08,E2 21196.08} C_VEL
LIN {X 0,Y 462.379,Z 315.73,A -85,B 0,C 180,E1 21194.227,E2 21194.227} C_VEL
LIN {X 0,Y 463.882,Z 318.802,A -85,B 0,C 180,E1 21193.985,E2 21193.985} C_VEL
LIN {X 0,Y 466.5,Z 337.303,A -85,B 0,C 180,E1 21193.272,E2 21193.272} C_VEL
LIN {X 0,Y 460.311,Z 528.611,A -85,B 0,C 180,E1 21189.785,E2 21189.785} C_VEL
LIN {X 0,Y 458.005,Z 605.738,A -85,B 0,C 180,E1 21188.385,E2 21188.385} C_VEL
LIN {X 0,Y 456.527,Z 628.104,A -85,B 0,C 180,E1 21187.767,E2 21187.767} C_VEL
LIN {X 0,Y 454.767,Z 649.266,A -85,B 0,C 180,E1 21186.962,E2 21186.962} C_VEL
LIN {X 0,Y 452.753,Z 669.729,A -85,B 0,C 180,E1 21185.973,E2 21185.973} C_VEL
LIN {X 0,Y 450.399,Z 690.574,A -85,B 0,C 180,E1 21184.707,E2 21184.707} C_VEL
LIN {X 0,Y 447.897,Z 710.605,A -85,B 0,C 180,E1 21183.231,E2 21183.231} C_VEL
LIN {X 0,Y 445.359,Z 729.884,A -85,B 0,C 180,E1 21181.538,E2 21181.538} C_VEL
LIN {X 0,Y 442.871,Z 748.308,A -85,B 0,C 180,E1 21179.63,E2 21179.63} C_VEL
LIN {X 0,Y 440.542,Z 765.051,A -85,B 0,C 180,E1 21177.579,E2 21177.579} C_VEL
LIN {X 0,Y 438.446,Z 780.473,A -85,B 0,C 180,E1 21175.385,E2 21175.385} C_VEL
LIN {X 0,Y 436.638,Z 794.633,A -85,B 0,C 180,E1 21173.051,E2 21173.051} C_VEL
LIN {X 0,Y 435.123,Z 807.323,A -85,B 0,C 180,E1 21170.582,E2 21170.582} C_VEL
LIN {X 0,Y 433.921,Z 818.679,A -85,B 0,C 180,E1 21167.983,E2 21167.983} C_VEL
LIN {X 0,Y 433.074,Z 828.242,A -85,B 0,C 180,E1 21165.395,E2 21165.395} C_VEL
LIN {X 0,Y 432.477,Z 836.383,A -85,B 0,C 180,E1 21162.672,E2 21162.672} C_VEL
LIN {X 0,Y 432.142,Z 842.64,A -85,B 0,C 180,E1 21159.992,E2 21159.992} C_VEL
LIN {X 0,Y 431.987,Z 847.227,A -85,B 0,C 180,E1 21157.312,E2 21157.312} C_VEL
LIN {X 0,Y 431.921,Z 850.445,A -85,B 0,C 180,E1 21154.513,E2 21154.513} C_VEL
LIN {X 0,Y 431.899,Z 852.209,A -85,B 0,C 180,E1 21151.723,E2 21151.723} C_VEL
LIN {X 0,Y 431.908,Z 852.347,A -85,B 0,C 180,E1 21149.07,E2 21149.07} C_VEL
LIN {X 0,Y 431.91,Z 851.121,A -85,B 0,C 180,E1 21146.282,E2 21146.282} C_VEL
LIN {X 0,Y 431.946,Z 848.454,A -85,B 0,C 180,E1 21143.62,E2 21143.62} C_VEL
LIN {X 0,Y 432.094,Z 843.904,A -85,B 0,C 180,E1 21140.677,E2 21140.677} C_VEL
LIN {X 0,Y 432.342,Z 838.792,A -85,B 0,C 180,E1 21138.256,E2 21138.256} C_VEL
LIN {X 0,Y 432.824,Z 831.136,A -85,B 0,C 180,E1 21135.552,E2 21135.552} C_VEL
LIN {X 0,Y 433.571,Z 822.173,A -85,B 0,C 180,E1 21132.969,E2 21132.969} C_VEL
LIN {X 0,Y 434.692,Z 810.582,A -85,B 0,C 180,E1 21130.236,E2 21130.236} C_VEL
LIN {X 0,Y 436.12,Z 797.338,A -85,B 0,C 180,E1 21127.63,E2 21127.63} C_VEL
LIN {X 0,Y 437.873,Z 782.426,A -85,B 0,C 180,E1 21125.155,E2 21125.155} C_VEL
LIN {X 0,Y 439.856,Z 766.341,A -85,B 0,C 180,E1 21122.885,E2 21122.885} C_VEL
LIN {X 0,Y 441.926,Z 749.313,A -85,B 0,C 180,E1 21120.848,E2 21120.848} C_VEL
LIN {X 0,Y 444.162,Z 730.91,A -85,B 0,C 180,E1 21118.968,E2 21118.968} C_VEL
LIN {X 0,Y 446.371,Z 712.063,A -85,B 0,C 180,E1 21117.327,E2 21117.327} C_VEL
LIN {X 0,Y 448.624,Z 691.533,A -85,B 0,C 180,E1 21115.83,E2 21115.83} C_VEL
LIN {X 0,Y 450.682,Z 670.698,A -85,B 0,C 180,E1 21114.573,E2 21114.573} C_VEL
LIN {X 0,Y 452.785,Z 647.422,A -85,B 0,C 180,E1 21113.442,E2 21113.442} C_VEL
LIN {X 0,Y 454.485,Z 625.511,A -85,B 0,C 180,E1 21112.612,E2 21112.612} C_VEL
LIN {X 0,Y 455.955,Z 601.714,A -85,B 0,C 180,E1 21111.965,E2 21111.965} C_VEL
LIN {X 0,Y 457.561,Z 546.139,A -85,B 0,C 180,E1 21110.933,E2 21110.933} C_VEL
LIN {X 0,Y 461.186,Z 440.969,A -85,B 0,C 180,E1 21108.924,E2 21108.924} C_VEL
LIN {X 0,Y 466.17,Z 340.527,A -85,B 0,C 180,E1 21106.826,E2 21106.826} C_VEL
LIN {X 0,Y 466.282,Z 335.102,A -85,B 0,C 180,E1 21106.68,E2 21106.68} C_VEL
LIN {X 0,Y 464.41,Z 316.81,A -85,B 0,C 180,E1 21105.847,E2 21105.847} C_VEL
LIN {X 0,Y 458.044,Z 302.274,A -85,B 0,C 180,E1 21104.29,E2 21104.29} C_VEL
LIN {X 0,Y 452.768,Z 291.374,A -85,B 0,C 180,E1 21102.728,E2 21102.728} C_VEL
LIN {X 0,Y 448.846,Z 284.002,A -85,B 0,C 180,E1 21101.253,E2 21101.253} C_VEL
LIN {X 0,Y 446.525,Z 279.565,A -85,B 0,C 180,E1 21100.075,E2 21100.075} C_VEL
LIN {X 0,Y 444.76,Z 275.695,A -85,B 0,C 180,E1 21098.681,E2 21098.681} C_VEL
LIN {X 0,Y 443.86,Z 273.548,A -85,B 0,C 180,E1 21096.899,E2 21096.899} C_VEL
LIN {X 0,Y 444.737,Z 272.914,A -85,B 0,C 180,E1 21095.296,E2 21095.296} C_VEL
LIN {X 0,Y 445.372,Z 273.325,A -85,B 0,C 180,E1 21094.697,E2 21094.697} C_VEL
LIN {X 0,Y 447.375,Z 276.797,A -85,B 0,C 180,E1 21093.292,E2 21093.292} C_VEL
LIN {X 0,Y 449.232,Z 278.589,A -85,B 0,C 180,E1 21092.483,E2 21092.483} C_VEL
LIN {X 0,Y 451.926,Z 282.732,A -85,B 0,C 180,E1 21091.437,E2 21091.437} C_VEL
LIN {X 0,Y 456.07,Z 289.033,A -85,B 0,C 180,E1 21090.172,E2 21090.172} C_VEL
LIN {X 0,Y 460.484,Z 296.12,A -85,B 0,C 180,E1 21089.045,E2 21089.045} C_VEL
LIN {X 0,Y 466.183,Z 306.39,A -85,B 0,C 180,E1 21087.782,E2 21087.782} C_VEL
LIN {X 0,Y 467.027,Z 308.499,A -85,B 0,C 180,E1 21087.597,E2 21087.597} C_VEL
LIN {X 0,Y 461.939,Z 401.449,A -85,B 0,C 180,E1 21085.627,E2 21085.627} C_VEL
LIN {X 0,Y 458.315,Z 497.152,A -85,B 0,C 180,E1 21083.764,E2 21083.764} C_VEL
LIN {X 0,Y 456.85,Z 541.57,A -85,B 0,C 180,E1 21082.9,E2 21082.9} C_VEL
LIN {X 0,Y 455.692,Z 563.957,A -85,B 0,C 180,E1 21082.234,E2 21082.234} C_VEL
LIN {X 0,Y 454.201,Z 584.451,A -85,B 0,C 180,E1 21081.396,E2 21081.396} C_VEL
LIN {X 0,Y 452.31,Z 605.374,A -85,B 0,C 180,E1 21080.309,E2 21080.309} C_VEL
LIN {X 0,Y 450.233,Z 624.96,A -85,B 0,C 180,E1 21079.055,E2 21079.055} C_VEL
LIN {X 0,Y 448,Z 643.486,A -85,B 0,C 180,E1 21077.604,E2 21077.604} C_VEL
LIN {X 0,Y 445.613,Z 661.22,A -85,B 0,C 180,E1 21075.955,E2 21075.955} C_VEL
LIN {X 0,Y 443.229,Z 678.062,A -85,B 0,C 180,E1 21074.102,E2 21074.102} C_VEL
LIN {X 0,Y 441.007,Z 692.971,A -85,B 0,C 180,E1 21072.174,E2 21072.174} C_VEL
LIN {X 0,Y 438.826,Z 707.39,A -85,B 0,C 180,E1 21069.973,E2 21069.973} C_VEL
LIN {X 0,Y 436.9,Z 720.463,A -85,B 0,C 180,E1 21067.629,E2 21067.629} C_VEL
LIN {X 0,Y 435.269,Z 732.17,A -85,B 0,C 180,E1 21065.141,E2 21065.141} C_VEL
LIN {X 0,Y 433.91,Z 742.935,A -85,B 0,C 180,E1 21062.379,E2 21062.379} C_VEL
LIN {X 0,Y 432.942,Z 752.133,A -85,B 0,C 180,E1 21059.472,E2 21059.472} C_VEL
LIN {X 0,Y 432.366,Z 759.169,A -85,B 0,C 180,E1 21056.688,E2 21056.688} C_VEL
LIN {X 0,Y 432.038,Z 765.578,A -85,B 0,C 180,E1 21053.357,E2 21053.357} C_VEL
LIN {X 0,Y 431.931,Z 769.559,A -85,B 0,C 180,E1 21050.408,E2 21050.408} C_VEL
LIN {X 0,Y 431.902,Z 771.814,A -85,B 0,C 180,E1 21047.569,E2 21047.569} C_VEL
LIN {X 0,Y 431.91,Z 772.489,A -85,B 0,C 180,E1 21044.838,E2 21044.838} C_VEL
LIN {X 0,Y 431.91,Z 771.657,A -85,B 0,C 180,E1 21042.07,E2 21042.07} C_VEL
LIN {X 0,Y 431.942,Z 769.156,A -85,B 0,C 180,E1 21039.118,E2 21039.118} C_VEL
LIN {X 0,Y 432.04,Z 765.06,A -85,B 0,C 180,E1 21036.257,E2 21036.257} C_VEL
LIN {X 0,Y 432.386,Z 758.73,A -85,B 0,C 180,E1 21033.051,E2 21033.051} C_VEL
LIN {X 0,Y 432.973,Z 751.389,A -85,B 0,C 180,E1 21030.234,E2 21030.234} C_VEL
LIN {X 0,Y 433.88,Z 742.591,A -85,B 0,C 180,E1 21027.506,E2 21027.506} C_VEL
LIN {X 0,Y 435.192,Z 731.842,A -85,B 0,C 180,E1 21024.786,E2 21024.786} C_VEL
LIN {X 0,Y 436.82,Z 719.9,A -85,B 0,C 180,E1 21022.266,E2 21022.266} C_VEL
LIN {X 0,Y 438.805,Z 706.333,A -85,B 0,C 180,E1 21019.85,E2 21019.85} C_VEL
LIN {X 0,Y 441.088,Z 691.301,A -85,B 0,C 180,E1 21017.573,E2 21017.573} C_VEL
LIN {X 0,Y 443.544,Z 675.073,A -85,B 0,C 180,E1 21015.491,E2 21015.491} C_VEL
LIN {X 0,Y 446.004,Z 658.274,A -85,B 0,C 180,E1 21013.669,E2 21013.669} C_VEL
LIN {X 0,Y 448.674,Z 639.057,A -85,B 0,C 180,E1 21011.904,E2 21011.904} C_VEL
LIN {X 0,Y 451.154,Z 619.838,A -85,B 0,C 180,E1 21010.428,E2 21010.428} C_VEL
LIN {X 0,Y 453.388,Z 600.055,A -85,B 0,C 180,E1 21009.185,E2 21009.185} C_VEL
LIN {X 0,Y 455.366,Z 579.392,A -85,B 0,C 180,E1 21008.132,E2 21008.132} C_VEL
LIN {X 0,Y 457.094,Z 557.656,A -85,B 0,C 180,E1 21007.269,E2 21007.269} C_VEL
LIN {X 0,Y 458.362,Z 536.544,A -85,B 0,C 180,E1 21006.66,E2 21006.66} C_VEL
LIN {X 0,Y 459.518,Z 501.859,A -85,B 0,C 180,E1 21005.999,E2 21005.999} C_VEL
LIN {X 0,Y 464.779,Z 332.237,A -85,B 0,C 180,E1 21002.937,E2 21002.937} C_VEL
LIN {X 0,Y 464.38,Z 325.738,A -85,B 0,C 180,E1 21002.75,E2 21002.75} C_VEL
LIN {X 0,Y 462.625,Z 318.643,A -85,B 0,C 180,E1 21002.4,E2 21002.4} C_VEL
LIN {X 0,Y 458.96,Z 310.359,A -85,B 0,C 180,E1 21001.8,E2 21001.8} C_VEL
LIN {X 0,Y 453.846,Z 302.158,A -85,B 0,C 180,E1 21001.015,E2 21001.015} C_VEL
LIN {X 0,Y 441.232,Z 283.559,A -85,B 0,C 180,E1 20999.009,E2 20999.009} C_VEL
LIN {X 0,Y 434.566,Z 274.118,A -85,B 0,C 180,E1 20997.882,E2 20997.882} C_VEL
LIN {X 0,Y 431.671,Z 269.934,A -85,B 0,C 180,E1 20997.374,E2 20997.374} C_VEL
LIN {X 0,Y 429.036,Z 265.936,A -85,B 0,C 180,E1 20996.899,E2 20996.899} C_VEL
LIN {X 0,Y 426.018,Z 262.24,A -85,B 0,C 180,E1 20996.371,E2 20996.371} C_VEL
LIN {X 0,Y 425.286,Z 259.762,A -85,B 0,C 180,E1 20996.191,E2 20996.191} C_VEL
LIN {X 0,Y 425.287,Z 259.76,A -85,B 0,C 180,E1 20992.388,E2 20992.388} C_VEL
LIN {X 0,Y 425.303,Z 259.754,A -85,B 0,C 180,E1 20988.648,E2 20988.648} C_VEL
LIN {X 0,Y 425.323,Z 259.757,A -85,B 0,C 180,E1 20984.848,E2 20984.848} C_VEL
LIN {X 0,Y 425.317,Z 259.751,A -85,B 0,C 180,E1 20980.978,E2 20980.978} C_VEL
LIN {X 0,Y 425.31,Z 259.754,A -85,B 0,C 180,E1 20977.159,E2 20977.159} C_VEL
LIN {X 0,Y 425.288,Z 259.756,A -85,B 0,C 180,E1 20973.371,E2 20973.371} C_VEL
LIN {X 0,Y 425.275,Z 259.752,A -85,B 0,C 180,E1 20969.597,E2 20969.597} C_VEL
LIN {X 0,Y 425.271,Z 259.747,A -85,B 0,C 180,E1 20965.822,E2 20965.822} C_VEL
LIN {X 0,Y 425.279,Z 259.75,A -85,B 0,C 180,E1 20962.028,E2 20962.028} C_VEL
LIN {X 0,Y 425.3,Z 259.75,A -85,B 0,C 180,E1 20958.337,E2 20958.337} C_VEL
LIN {X 0,Y 425.319,Z 259.749,A -85,B 0,C 180,E1 20954.534,E2 20954.534} C_VEL
LIN {X 0,Y 425.312,Z 259.751,A -85,B 0,C 180,E1 20950.643,E2 20950.643} C_VEL
LIN {X 0,Y 425.288,Z 259.757,A -85,B 0,C 180,E1 20946.884,E2 20946.884} C_VEL
LIN {X 0,Y 425.27,Z 259.759,A -85,B 0,C 180,E1 20943.167,E2 20943.167} C_VEL
LIN {X 0,Y 425.263,Z 259.761,A -85,B 0,C 180,E1 20939.369,E2 20939.369} C_VEL
LIN {X 0,Y 425.268,Z 259.763,A -85,B 0,C 180,E1 20935.608,E2 20935.608} C_VEL
LIN {X 0,Y 425.283,Z 259.762,A -85,B 0,C 180,E1 20931.808,E2 20931.808} C_VEL
LIN {X 0,Y 425.308,Z 259.753,A -85,B 0,C 180,E1 20928.116,E2 20928.116} C_VEL
LIN {X 0,Y 425.299,Z 259.755,A -85,B 0,C 180,E1 20924.281,E2 20924.281} C_VEL
LIN {X 0,Y 425.283,Z 259.762,A -85,B 0,C 180,E1 20920.454,E2 20920.454} C_VEL
LIN {X 0,Y 425.257,Z 259.763,A -85,B 0,C 180,E1 20916.835,E2 20916.835} C_VEL
LIN {X 0,Y 425.253,Z 259.762,A -85,B 0,C 180,E1 20913.054,E2 20913.054} C_VEL
LIN {X 0,Y 425.261,Z 259.76,A -85,B 0,C 180,E1 20909.275,E2 20909.275} C_VEL
LIN {X 0,Y 425.286,Z 259.752,A -85,B 0,C 180,E1 20905.629,E2 20905.629} C_VEL
LIN {X 0,Y 425.307,Z 259.753,A -85,B 0,C 180,E1 20901.787,E2 20901.787} C_VEL
LIN {X 0,Y 425.288,Z 259.756,A -85,B 0,C 180,E1 20897.935,E2 20897.935} C_VEL
LIN {X 0,Y 425.255,Z 259.759,A -85,B 0,C 180,E1 20894.29,E2 20894.29} C_VEL
LIN {X 0,Y 425.242,Z 259.757,A -85,B 0,C 180,E1 20890.566,E2 20890.566} C_VEL
LIN {X 0,Y 425.241,Z 259.76,A -85,B 0,C 180,E1 20886.75,E2 20886.75} C_VEL
LIN {X 0,Y 425.251,Z 259.764,A -85,B 0,C 180,E1 20882.963,E2 20882.963} C_VEL
LIN {X 0,Y 425.288,Z 259.763,A -85,B 0,C 180,E1 20879.325,E2 20879.325} C_VEL
LIN {X 0,Y 425.292,Z 259.759,A -85,B 0,C 180,E1 20875.404,E2 20875.404} C_VEL
LIN {X 0,Y 425.285,Z 259.757,A -85,B 0,C 180,E1 20871.617,E2 20871.617} C_VEL
LIN {X 0,Y 425.259,Z 259.76,A -85,B 0,C 180,E1 20867.92,E2 20867.92} C_VEL
LIN {X 0,Y 425.248,Z 259.761,A -85,B 0,C 180,E1 20864.311,E2 20864.311} C_VEL
LIN {X 0,Y 425.256,Z 259.76,A -85,B 0,C 180,E1 20860.495,E2 20860.495} C_VEL
LIN {X 0,Y 425.278,Z 259.755,A -85,B 0,C 180,E1 20856.814,E2 20856.814} C_VEL
LIN {X 0,Y 425.303,Z 259.755,A -85,B 0,C 180,E1 20852.995,E2 20852.995} C_VEL
LIN {X 0,Y 425.309,Z 259.756,A -85,B 0,C 180,E1 20849.097,E2 20849.097} C_VEL
LIN {X 0,Y 425.287,Z 259.759,A -85,B 0,C 180,E1 20845.322,E2 20845.322} C_VEL
LIN {X 0,Y 425.295,Z 259.86,A -85,B 0,C 180,E1 20843.378,E2 20843.378} C_VEL
LIN {X 0,Y 426.607,Z 263.246,A -85,B 0,C 180,E1 20842.793,E2 20842.793} C_VEL
LIN {X 0,Y 427.69,Z 265.285,A -85,B 0,C 180,E1 20842.397,E2 20842.397} C_VEL
LIN {X 0,Y 434.17,Z 278.418,A -85,B 0,C 180,E1 20840.019,E2 20840.019} C_VEL
LIN {X 0,Y 442.422,Z 295.875,A -85,B 0,C 180,E1 20837.158,E2 20837.158} C_VEL
LIN {X 0,Y 454.073,Z 315.065,A -85,B 0,C 180,E1 20835.221,E2 20835.221} C_VEL
LIN {X 0,Y 458.271,Z 322.661,A -85,B 0,C 180,E1 20834.538,E2 20834.538} C_VEL
LIN {X 0,Y 460.477,Z 338.895,A -85,B 0,C 180,E1 20833.906,E2 20833.906} C_VEL
LIN {X 0,Y 453.846,Z 531.206,A -85,B 0,C 180,E1 20830.345,E2 20830.345} C_VEL
LIN {X 0,Y 451.476,Z 605.321,A -85,B 0,C 180,E1 20828.975,E2 20828.975} C_VEL
LIN {X 0,Y 449.897,Z 627.955,A -85,B 0,C 180,E1 20828.343,E2 20828.343} C_VEL
LIN {X 0,Y 448.05,Z 648.997,A -85,B 0,C 180,E1 20827.531,E2 20827.531} C_VEL
LIN {X 0,Y 445.939,Z 669.39,A -85,B 0,C 180,E1 20826.531,E2 20826.531} C_VEL
LIN {X 0,Y 443.447,Z 690.181,A -85,B 0,C 180,E1 20825.253,E2 20825.253} C_VEL
LIN {X 0,Y 440.926,Z 709.32,A -85,B 0,C 180,E1 20823.826,E2 20823.826} C_VEL
LIN {X 0,Y 438.236,Z 728.708,A -85,B 0,C 180,E1 20822.112,E2 20822.112} C_VEL
LIN {X 0,Y 435.596,Z 747.189,A -85,B 0,C 180,E1 20820.176,E2 20820.176} C_VEL
LIN {X 0,Y 433.1,Z 764,A -85,B 0,C 180,E1 20818.094,E2 20818.094} C_VEL
LIN {X 0,Y 430.754,Z 780.379,A -85,B 0,C 180,E1 20815.724,E2 20815.724} C_VEL
LIN {X 0,Y 428.852,Z 794.45,A -85,B 0,C 180,E1 20813.348,E2 20813.348} C_VEL
LIN {X 0,Y 427.258,Z 807.103,A -85,B 0,C 180,E1 20810.835,E2 20810.835} C_VEL
LIN {X 0,Y 425.995,Z 818.38,A -85,B 0,C 180,E1 20808.188,E2 20808.188} C_VEL
LIN {X 0,Y 425.074,Z 828.301,A -85,B 0,C 180,E1 20805.413,E2 20805.413} C_VEL
LIN {X 0,Y 424.497,Z 835.937,A -85,B 0,C 180,E1 20802.79,E2 20802.79} C_VEL
LIN {X 0,Y 424.138,Z 842.585,A -85,B 0,C 180,E1 20799.908,E2 20799.908} C_VEL
LIN {X 0,Y 423.986,Z 847.344,A -85,B 0,C 180,E1 20797.179,E2 20797.179} C_VEL
LIN {X 0,Y 423.921,Z 850.446,A -85,B 0,C 180,E1 20794.463,E2 20794.463} C_VEL
LIN {X 0,Y 423.9,Z 852.175,A -85,B 0,C 180,E1 20791.756,E2 20791.756} C_VEL
LIN {X 0,Y 423.908,Z 852.321,A -85,B 0,C 180,E1 20789.053,E2 20789.053} C_VEL
LIN {X 0,Y 423.911,Z 851.039,A -85,B 0,C 180,E1 20786.212,E2 20786.212} C_VEL
LIN {X 0,Y 423.947,Z 848.368,A -85,B 0,C 180,E1 20783.635,E2 20783.635} C_VEL
LIN {X 0,Y 424.087,Z 843.859,A -85,B 0,C 180,E1 20780.773,E2 20780.773} C_VEL
LIN {X 0,Y 424.363,Z 838.217,A -85,B 0,C 180,E1 20778.17,E2 20778.17} C_VEL
LIN {X 0,Y 424.855,Z 830.555,A -85,B 0,C 180,E1 20775.414,E2 20775.414} C_VEL
LIN {X 0,Y 425.622,Z 821.572,A -85,B 0,C 180,E1 20772.782,E2 20772.782} C_VEL
LIN {X 0,Y 426.724,Z 810.609,A -85,B 0,C 180,E1 20770.137,E2 20770.137} C_VEL
LIN {X 0,Y 428.194,Z 797.498,A -85,B 0,C 180,E1 20767.482,E2 20767.482} C_VEL
LIN {X 0,Y 430.006,Z 782.727,A -85,B 0,C 180,E1 20764.963,E2 20764.963} C_VEL
LIN {X 0,Y 431.988,Z 767.225,A -85,B 0,C 180,E1 20762.722,E2 20762.722} C_VEL
LIN {X 0,Y 434.162,Z 750.242,A -85,B 0,C 180,E1 20760.623,E2 20760.623} C_VEL
LIN {X 0,Y 436.534,Z 731.688,A -85,B 0,C 180,E1 20758.671,E2 20758.671} C_VEL
LIN {X 0,Y 438.937,Z 712.302,A -85,B 0,C 180,E1 20756.936,E2 20756.936} C_VEL
LIN {X 0,Y 441.234,Z 692.37,A -85,B 0,C 180,E1 20755.45,E2 20755.45} C_VEL
LIN {X 0,Y 443.58,Z 670.269,A -85,B 0,C 180,E1 20754.077,E2 20754.077} C_VEL
LIN {X 0,Y 445.733,Z 647.938,A -85,B 0,C 180,E1 20752.965,E2 20752.965} C_VEL
LIN {X 0,Y 447.615,Z 625.4,A -85,B 0,C 180,E1 20752.084,E2 20752.084} C_VEL
LIN {X 0,Y 449.199,Z 601.742,A -85,B 0,C 180,E1 20751.42,E2 20751.42} C_VEL
LIN {X 0,Y 450.554,Z 561.284,A -85,B 0,C 180,E1 20750.631,E2 20750.631} C_VEL
LIN {X 0,Y 454.224,Z 460.702,A -85,B 0,C 180,E1 20748.673,E2 20748.673} C_VEL
LIN {X 0,Y 459.105,Z 366.599,A -85,B 0,C 180,E1 20746.668,E2 20746.668} C_VEL
LIN {X 0,Y 460.863,Z 337.027,A -85,B 0,C 180,E1 20745.986,E2 20745.986} C_VEL
LIN {X 0,Y 459.413,Z 320.912,A -85,B 0,C 180,E1 20745.217,E2 20745.217} C_VEL
LIN {X 0,Y 453.815,Z 307.15,A -85,B 0,C 180,E1 20743.687,E2 20743.687} C_VEL
LIN {X 0,Y 449.464,Z 297.67,A -85,B 0,C 180,E1 20742.251,E2 20742.251} C_VEL
LIN {X 0,Y 446.05,Z 290.702,A -85,B 0,C 180,E1 20740.801,E2 20740.801} C_VEL
LIN {X 0,Y 444.2,Z 286.794,A -85,B 0,C 180,E1 20739.738,E2 20739.738} C_VEL
LIN {X 0,Y 442.758,Z 283.204,A -85,B 0,C 180,E1 20738.392,E2 20738.392} C_VEL
LIN {X 0,Y 442.245,Z 281.189,A -85,B 0,C 180,E1 20736.619,E2 20736.619} C_VEL
LIN {X 0,Y 443.382,Z 280.813,A -85,B 0,C 180,E1 20734.993,E2 20734.993} C_VEL
LIN {X 0,Y 445.304,Z 284.379,A -85,B 0,C 180,E1 20733.484,E2 20733.484} C_VEL
LIN {X 0,Y 446.798,Z 285.972,A -85,B 0,C 180,E1 20732.773,E2 20732.773} C_VEL
LIN {X 0,Y 450.07,Z 291.233,A -85,B 0,C 180,E1 20731.451,E2 20731.451} C_VEL
LIN {X 0,Y 453.394,Z 296.697,A -85,B 0,C 180,E1 20730.385,E2 20730.385} C_VEL
LIN {X 0,Y 457.334,Z 303.439,A -85,B 0,C 180,E1 20729.324,E2 20729.324} C_VEL
